# B&R Automation Studio project 8238 (part 19)

### history.Pkg_mnParam.txt
```
0.2.0	18.8.2011	- Import-Verzeichnis wird im Hochlauf gelöscht
			- Es werden auch REAL-Parameter unterstützt. (not tested)
0.3.0	24.8.2011	- IP-CSV-Rowtype ergänzt. (90)
0.4.0	01.09.2011	- Info_typ geändert. Es wird jetzt auch ausgegeben, welcher Container geändert wurde
0.5.0	20.09.2011	- mnParamStat und mnParamStatAd ergänzt.
			  Kapselung von Stati. z.B. xParamOK, dtExportContent
0.6.0	07.10.2011	- Maschinennummer wird aus _mnr.csv gelesen und in die _Info_-Struktur geschrieben
0.6.1	18.11.2011	- Liefert jetzt eine Fehlermeldung, wenn die zu importierende Datei keine Maschinennummer enthält
0.6.2	28.11.2011	- mnParamLib : mnParam_WritePVNum. UDINT wurde als UINT behandelt.
0.7.0	20.10.2011	- Umstellung auf AS 3.0.90
					- Berücksichtigung von WSTRING
					- utfMachineNumber und xParamOK in das IFmnParam.Out
0.8.0	20.12.2011	- Logging in das Logbuch der AR verlegt.
					- EXIT hinzugefügt.
					- Fehler im Init-Up behoben.
0.8.1	22.12.2011	- Severity für Log angepasst
0.8.2	02.01.2012	- Initialisierung der Text-Zeilen in GetCsvDat
					- Sprachdefinition ist 248, nicht 247
0.9.0	03.01.2012	- Packetversion in mnParamStatAd
0.9.1	10.01.2012	- Kommentar der Package-Version im Export wird dynamisch gelesen
0.10.0	18.01.2012	- Textzeilen werden jetzt mit bis zu 63 Zeichen ausgelesen
0.11.0	13.02.2012	- Speicherloch in der Initialisierung beseitigt. Beim Importieren vorhandener Datencontainer wurde Speicher nicht mehr frei gegeben.
0.11.1	15.02.2012	- Weiterentwicklung: Speicheroptimierung. Automatische Berechnung der Größe der Speicherpartition.
		16.02.2012	- Einführung von Funktionsbausteinen für Standardfunktionen.
					- Schreiben eines Inhaltsverzeichnisses von CSV-Datencontainerdateien im Exportverzeichnis
		17.02.2012	- Unit ist UINT
0.11.2	22.02.2012	- Helptext wurde auf 63 Zeichen begrenzt
					- Kompatibel zu hlKanLink 0.94.0
0.12.0	06.03.2012	- Kompatibel zu mnTest
0.12.1	08.03.2012	- Bugfix Editliste füllen
0.13.0	15.03.2012	- Editliste wird mit umgerechneten Werten gefüllt.
0.13.1	15.03.2012	- Ergänzt um die Anzahl der Nachkommastellen
					- Datenmodell erweitert um RefVisible und RefText
0.13.2	20.03.2012	- Abhängigkeiten ergänzt
0.13.9	20.03.2012	- Zwischenstand - Weiterentwicklung mnParam
0.14.0	21.03.2012	- Save-Editor und Delete indirect container implementiert. Bugfix im Delete Algorithmus auch für mnParamCmd
0.15.0	22.03.2012	- Zwischenversion. Es wird jetzt für das Edit-Feld nach Parameterindex, und nicht nach Container-Index gesucht.
					- Letzter Parameter eines Containers wurde nicht ausgelesen
					- Massenimport implementiert
					- Restore ist möglich
0.15.1	23.03.2012	- Maschinennummer des Datencontainers wird jetzt auch im Init-Up überprüft.
					- Die Überprüfung der Maschinennummer im zyklischen Teil kann applikativ deaktiviert werden.
					- Logger implementiert
					- Backup und Restore implementiert
0.16.0	23.03.2012	- Release
0.16.1	27.03.2012	- Bugfix: Container wurden im Init-Up nicht eingelesen
0.16.2	27.03.2012	- Weiterentwicklung
0.17.0	28.03.2012	- Namensliste für Instanzen kann gefüllt werden
					- Instanz NEU und KOPIEREN ist implementiert
0.17.1	29.03.2012	- Bugfix. Save Editor. Letzter Eintrag wurde nicht gesichert
0.18.0	29.03.2012	- Kategorie-Programm-Zuordnung ergänzt
0.18.1	30.03.2012	- Kategorie-Programm-Zuordnung um Kategorienamen erweitert
0.18.2	02.04.2012	- Kategoriedaten erweitert
0.19.0	03.04.2012	- Warnungen bei Importfehler
		04.04.2012	- _Info_ wird nicht mehr unterstützt
					- Bugfix: TOC wurde beim Import vom PC nicht aktualisiert
0.20.0	05.04.2012	- Die Quelle zum Füllen der Namensliste wird nur initial von den Konstanten übernommen.
					  Per Befehl kann die Quelle geändert werden.
0.20.1	10.04.2012	- Wenn die Dateien im Exportverzeichnis gelöscht wurden, hat der Parametermanager diese nicht
					  neu angelegt.
0.20.2	11.04.2012	- Maschinennummer mit Länge 0 wird als Fehler abgefangen
0.20.3	11.04.2012	- Ungültige Maschinennummer "dummy" als Konstante MNPARAM_INVALID_MACHINENO eingeführt
0.20.4	13.04.2012	- Warnung wird angezeigt, wenn der Parametermanager nicht bereit ist.
0.20.5	16.04.2012	- Beim Füllen des Editors, wurden die Parameter für die Namensliste zurückgesetzt
0.20.6	17.04.2012	- Es konnten keine Instanzen aus dem Editor gesichert werden. Der Pointer auf die StrucRoot wurde nicht ermittelt.
0.20.7	18.04.2012  - Instanz-Datenobjekte werden im Init teilweise wieder gelöscht.
					- In der Instanznamensliste werden noch die Instanznummern vorangestellt
0.21.0	23.04.2012	- Wir create instance oder copy instance eine negative Instanznummer übergeben, wird die nächste freie Instanz angelegt
					- Bei Fill Namelist wird automatisch die Category-Program-Cache-Liste aktualisiert
0.21.1	23.04.2012	- Copy hat nicht funktioniert
0.22.0	11.05.2012	- Restore lädt auch den cpcache
0.23.0	04.06.2012	- Im InitUp werden beim Importieren der Container auf jeden Falle vorher alle Daten auf Default gesetzt.
					- Wird nach dem Hochlauf ein USB-Stick mit dem Unterverzeichnis SetupKG erkannt, dann wird das Userverzeichnis entsprechend
					  überschrieben
					- Die Struktur "Machinestate" wird nicht mehr unterstützt
0.24.0 12.06.2012	- Beim Import von Parametern werden numerische Parameter auf ihre min- und max-Werte begrenzt.
					- Hilfstexte für Parameter auf 255 Zeichen erweitert.
					- Im Parametereditor kann nun gesteuert werden, ob Funktions- und Instanztexte in den Parametertext eingefügt werden.
					  Zusätzlich wird der Funktionstext und Instanztext zum Parameter separat ausgegeben. Parameter können nach Funktionen
					  gefiltert werden
0.24.1	26.06.2012	- Warnung unterdrückt
0.24.2	17.07.2012	- Filehandles wurden nach FileCreate nicht freigegeben.
0.24.3	03.09.2012	- Bugfix: Bug 835 - Kopierte Datencontainer sind schreibgeschützt. Behoben
0.25.0	06.09.2012	- Erweiterung Bug 821: Neue Konstante: MNPARAM_REQMISSINGMNO vom Typ USINT
					  0 : Wenn die Datei _mnr.csv fehlt, wird die Maschinennummer "dummy" gesetzt.
					  1 : Wenn die Datei _mnr.csv fehlt, erwartet der Parametermanager über das Interface IFmnParam
					  	  das Setzen der Maschinennummer in IFmnParam.In.utfSetMachineNumber. Danach muss die Strukturvariable
						  IFmnParam.In.xSetMachnineNumber auf TRUE gesetzt werden. Die _mnr.csv wird erzeugt und die Steuerung wird
						  neu gestartet.
```

### CfgMsgStat.mnParam.txt
```
;****************************
; Parameter Manager
;*****************************
00001, 00001, 00000, 00000;
00001, 00002, 00000, 00000;
00001, 00003, 00000, 00000;
00001, 00004, 00000, 00000;
00001, 00005, 00000, 00000;
00001, 00006, 00000, 00000;
00001, 00007, 00000, 00000;
00001, 00009, 00000, 00000;
00001, 20000, 00000, 00000;
```

### Package Logical/Standard/Kanlink/KGFramework/Pkg_mnTxt - Text-Manager

### Pkg_mnTxt.typ - Global data types
```iecst
(********************************************************************
 * COPYRIGHT -- Herbert Kannegiesser GmbH
 ********************************************************************
 * Package: Pkg_mnTxt
 * File: Pkg_mnTxt.typ
 * Author: hunholz
 * Created: November 25, 2011
 ********************************************************************
 * Data types of package Pkg_mnTxt
 ********************************************************************)
(*Interface*)

TYPE
	IFmnTxt_Typ : 	STRUCT
		In : IFmnTxt_In_Typ;
		Out : IFmnTxt_Out_Typ;
	END_STRUCT;
	IFmnTxt_Out_Typ : 	STRUCT
		wSelectedLanguage : UINT; (*Aktive Sprache*)
		wSelectLanguageStatus : UINT; (*0 - Sprache gültig, nur dann sind auch die Pointer auf die Texte gültig
60000..65000 - Fehler
65535 - Sprache wird geladen*)
		wLCIDs : ARRAY[0..MNTXT_MAX_IDX_LCID]OF UINT;
		wCntLCID : UINT;
		wCntInstanceTxt : UINT := 0;
		wCntFunctionTxt : UINT := 0;
		wCntParamTxt : UINT := 0;
		wCntParamHlpTxt : UINT := 0;
		wCntMessageTxt : UINT := 0;
		wCntMessageHlpTxt : UINT := 0;
		ptrInstanceTxtList : UDINT; (*Zeigt auf das Datenobjekt _mnTxtI, Zeilen vom Typ mnTxt_TxtLine_Typ*)
		ptrFunctionTxtList : UDINT; (*Zeigt auf das Datenobjekt _mnTxtF, Zeilen vom Typ mnTxt_TxtLine_Typ*)
		ptrParamTxtList : UDINT; (*Zeigt auf das Datenobjekt _mnTxtP, Zeilen vom Typ mnTxt_TxtLine_Typ*)
		ptrParamHelpTxtList : UDINT; (*Zeigt auf das Datenobjekt _mnTxtPh, Zeilen vom Typ mnTxt_HelpTxtLine_Typ*)
		ptrMessageTxtList : UDINT; (*Zeigt auf das Datenobjekt _mnTxtM, Zeilen vom Typ mnTxt_TxtLine_Typ*)
		ptrMessageHelpTxtList : UDINT; (*Zeigt auf das Datenobjekt _mnTxtMh, Zeilen vom Typ mnTxt_HelpTxtLine_Typ*)
	END_STRUCT;
	IFmnTxt_In_Typ : 	STRUCT
		wSelectLanguage : UINT; (*LCID der Sprache, die genutzt werden soll*)
	END_STRUCT;
END_TYPE

(*Parameter*)

TYPE
	mnTxtPar_Typ : 	STRUCT
		Mac : mnTxtPar_Mac_Typ; (*Maschinenparameter*)
	END_STRUCT;
	mnTxtPar_Mac_Typ : 	STRUCT
		wStartUpLanguage : UINT := 0; (*Die Sprache ist remanent. Ist hier ein Wert > 0 gewählt, wird diese Sprache beim Einschalten immer geladen.*)
	END_STRUCT;
END_TYPE

(*Status*)

TYPE
	mnTxtStatAd_Typ : 	STRUCT
		sPkgVersion : STRING[10];
	END_STRUCT;
END_TYPE

(*Öffentliche Typen*)

TYPE
	mnTxt_TxtLine_Typ : 	STRUCT
		wFunctionID : UINT; (*Funktions-Identifier*)
		wNumber : UINT; (*Textnummer*)
		wInstance : UINT; (*Instanznummer, um kompatibel zu mnMsg zu sein*)
		utfText : WSTRING[63]; (*Eigentlicher Text*)
	END_STRUCT;
	mnTxt_HelpTxtLine_Typ : 	STRUCT
		wFunctionID : UINT; (*Funktions-Identifier*)
		wNumber : UINT; (*Textnummer*)
		wInstance : UINT; (*Instanznummer, um kompatibel zu mnMsg zu sein*)
		utfText : WSTRING[255]; (*Eigentlicher Hilfstext*)
	END_STRUCT;
END_TYPE
```

### Pkg_mnTxt.var - Global variables
```iecst
(********************************************************************
 * COPYRIGHT -- Herbert Kannegiesser GmbH
 ********************************************************************
 * Package: Pkg_mnTxt
 * File: Pkg_mnTxt.var
 * Author: hunholz
 * Created: November 25, 2011
 ********************************************************************
 * Variables of package Pkg_mnTxt
 ********************************************************************)
(*KONSTANTEN*)
VAR CONSTANT
	MNTXT_DATOBJNAME_INSTXT : STRING[11] := '_mnTxtI'; (*Name des Datenmoduls, in dem die Instanztexte abgelegt sind*)
	MNTXT_DATOBJNAME_FUNTXT : STRING[11] := '_mnTxtF'; (*Name des Datenmoduls, in dem die Funktionstexte abgelegt sind*)
	MNTXT_DATOBJNAME_PARTXT : STRING[11] := '_mnTxtP'; (*Name des Datenmoduls, in dem die Parametertexte abgelegt sind*)
	MNTXT_DATOBJNAME_PARHELPTXT : STRING[11] := '_mnTxtPh'; (*Name des Datenmoduls, in dem die Parameterhilfstexte abgelegt sind*)
	MNTXT_DATOBJNAME_MSGTXT : STRING[11] := '_mnTxtM'; (*Name des Datenmoduls, in dem die Meldungstexte abgelegt sind*)
	MNTXT_DATOBJNAME_MSGHELPTXT : STRING[11] := '_mnTxtMh'; (*Name des Datenmoduls, in dem die Meldungshilfstexte abgelegt sind*)
END_VAR
(*-- LCID --*)
VAR CONSTANT
	MNTXT_LCID_GERMAN : UINT := 1031; (*LCID German*)
	MNTXT_LCID_ENGLISH_US : UINT := 1033; (*LCID English USA*)
END_VAR
(*-- Stati --*)
VAR CONSTANT
	MNTXT_STAT_OK : UINT := 0;
	MNTXT_STAT_NOLANGUAGE : UINT := 1; (*Keine gültige Sprache geladen*)
	MNTXT_STAT_INIT : UINT := 100;
	MNTXT_STAT_ERRDATOBJ : UINT := 60000; (*Datenobjekte für Texte konnten nicht erstellt werden.*)
	MNTXT_STAT_ERRMSGCFG : UINT := 60001; (*Message-Config Fehler*)
	MNTXT_STAT_ERRMEM : UINT := 60002; (*Speicher nicht allokierbar oder nicht ausreichend*)
	MNTXT_STAT_ERRLCID : UINT := 60003; (*Fehler beim laden von LCID.csv*)
	MNTXT_STAT_ERRFUNCTIONTXT : UINT := 60004;
	MNTXT_STAT_ERRINSTANCETXT : UINT := 60005;
	MNTXT_STAT_ERRMESSAGETXT : UINT := 60006;
	MNTXT_STAT_ERRPARAMTXT : UINT := 60007;
	MNTXT_STAT_LOADING : UINT := 65535;
END_VAR
(*Interface*)
VAR
	IFmnTxt : IFmnTxt_Typ;
END_VAR
(*Status*)
VAR
	mnTxtStatAd : mnTxtStatAd_Typ;
END_VAR
(*Parameter*)
VAR
	mnTxtPar : mnTxtPar_Typ;
END_VAR
```

### Program Logical/Standard/Kanlink/KGFramework/Pkg_mnTxt/mnTxt (IEC) - Text-Manager

#### mnTxtCyclic.st - Cyclic code
```iecst
(********************************************************************
 * COPYRIGHT -- Herbert Kannegiesser GmbH
 ********************************************************************
 * Program: mnTxt
 * File: mnTxtCyclic.st
 * Author: hunholz
 * Created: November 25, 2011
 ********************************************************************
 * Implementation of program mnTxt
 ********************************************************************)

PROGRAM _CYCLIC

	// Auf Sprachwechsel reagieren, bzw. letzte Sprache laden

	IF _xInitOK THEN

		IF IFmnTxt.Out.wSelectLanguageStatus = MNTXT_STAT_OK THEN

			// Sprache kann neu gewählt werden
			IF _wActLCID <> IFmnTxt.In.wSelectLanguage AND IFmnTxt.In.wSelectLanguage <> 0 THEN

				_wIdxLCID := 0;

				REPEAT

					IF IFmnTxt.In.wSelectLanguage = IFmnTxt.Out.wLCIDs[_wIdxLCID] THEN

						_wActLCID := IFmnTxt.In.wSelectLanguage;

						IFmnTxt.Out.wSelectedLanguage := _wActLCID;
						IFmnTxt.Out.wSelectLanguageStatus := MNTXT_STAT_LOADING;
						_LoadState := _ls_load_functiontxt_01;

					END_IF

					_wIdxLCID := _wIdxLCID + 1;

					UNTIL
					_wActLCID = IFmnTxt.In.wSelectLanguage OR _wIdxLCID >= IFmnTxt.Out.wCntLCID OR _wIdxLCID > MNTXT_MAX_IDX_LCID
				END_REPEAT

			END_IF

		ELSIF IFmnTxt.Out.wSelectLanguageStatus = MNTXT_STAT_NOLANGUAGE THEN

			IF _LoadState = _ls_idle THEN

				// Sprache erstmals laden
				IF _wActLCID = 0 THEN

					IF _xGermanExist THEN

						_wActLCID := MNTXT_LCID_GERMAN;

					ELSE

						_wActLCID := IFmnTxt.Out.wLCIDs[0];

					END_IF

				END_IF

				IFmnTxt.Out.wSelectedLanguage := _wActLCID;
				IFmnTxt.Out.wSelectLanguageStatus := MNTXT_STAT_LOADING;
				_LoadState := _ls_load_functiontxt_01;

			END_IF

		END_IF

	END_IF

	// Zyklusbegrenzung zurücksetzen

	_lCycleCounter := 0;

	// Statemachine

	CASE _LoadState OF

		_ls_idle:

		// Grundzustand, nichts tun

		//###########################################################################################
		// FUNKTIONSTEXTE LADEN
		//###########################################################################################

		_ls_load_functiontxt_01:

			// Nachsehen, ob Funktionstexte existieren

			IFmnTxt.Out.wCntFunctionTxt := 0;

			IF MNTXT_LOAD_FUNCTIONTEXT AND _CheckDoFunc.doId <> 0 THEN

				IF MNTXT_ENABLE_LANSPECRESOURCE = 1 THEN

					_sLCID := UINT_TO_STRING(_wActLCID);
					_sPath := CONCAT('Language\Function',_sLCID);
					_sPath := CONCAT(_sPath,'.csv');

				ELSE

					_sPath := 'Language\Function.csv';

				END_IF

				_FileInfo(enable := TRUE, pDevice := ADR(KG_DEVICE_COMPACTFLASH), pName := ADR(_sPath), pInfo := ADR(_fiFileInfo));

				IF _FileInfo.status = ERR_OK THEN

					_LoadState := _ls_load_functiontxt_02;

				ELSIF _FileInfo.status <> ERR_FUB_BUSY THEN

					_LoadState := _ls_load_instancetxt_01;

				END_IF

			ELSE

				_LoadState := _ls_load_instancetxt_01;

			END_IF

		_ls_load_functiontxt_02:

			// Speicher zum Parsen der Funktionstexte allokieren
			_MemPartAlloc(enable := TRUE, ident := _MemPartCreate.ident, len := _fiFileInfo.size-SIZEOF(KGBOM) );

			IF _MemPartAlloc.status = ERR_OK THEN

				_lAdrFile := _MemPartAlloc.mem;
				_LoadState := _ls_load_functiontxt_03;

			ELSIF _MemPartAlloc.status <> ERR_FUB_BUSY THEN

				IFmnTxt.Out.wSelectLanguageStatus := MNTXT_STAT_ERRMEM;
				_LoadState := _ls_error;

			END_IF

		_ls_load_functiontxt_03:

			_FileOpen(enable := TRUE, pDevice := ADR(KG_DEVICE_COMPACTFLASH), pFile := ADR(_sPath), mode := fiREAD_ONLY);

			IF _FileOpen.status = ERR_OK THEN

				_LoadState := _ls_load_functiontxt_04;

			ELSIF _FileOpen.status <> ERR_FUB_BUSY THEN

				IFmnTxt.Out.wSelectLanguageStatus := MNTXT_STAT_ERRFUNCTIONTXT;
				_LoadState := _ls_error;

			END_IF

		_ls_load_functiontxt_04:

			_FileRead(enable := TRUE, ident := _FileOpen.ident, offset := SIZEOF(KGBOM),pDest := _lAdrFile, len :=  _fiFileInfo.size-SIZEOF(KGBOM) );

			IF _FileRead.status <> ERR_FUB_BUSY THEN

				_LoadState := _ls_load_functiontxt_05;

			END_IF

		_ls_load_functiontxt_05:

			_FileClose(enable := TRUE, ident := _FileOpen.ident);

			IF _FileClose.status <> ERR_FUB_BUSY THEN

				IF _FileRead.status = ERR_OK THEN

					_LoadState := _ls_load_functiontxt_06;

				ELSE
					IFmnTxt.Out.wSelectLanguageStatus := MNTXT_STAT_ERRFUNCTIONTXT;
					_LoadState := _ls_error;

				END_IF

			END_IF

		_ls_load_functiontxt_06:

			// Zeilen in der Datei zählen und Startadressen ermitteln

			_CountLines.enable := TRUE;
			_CountLines.pFile := _lAdrFile;
			_CountLines.FileSize := _fiFileInfo.size - SIZEOF(KGBOM);
			_CountLines.MaxLines := MNTXT_MAXPARSELINES;
			_CountLines.pAdresses := _lAdrLineAdress;
			_CountLines.pLens := _lAdrLineLen;

			_CountLines();

			IF _CountLines.status = ERR_OK THEN

				_LoadState := _ls_load_functiontxt_07;

				_wStartLine := 1;
				_wIdxFunctionTxt := 0;
				_GetCsvDat.enable := TRUE;

			ELSE

				IFmnTxt.Out.wSelectLanguageStatus := MNTXT_STAT_ERRFUNCTIONTXT;
				_LoadState := _ls_error;

			END_IF

		_ls_load_functiontxt_07:

			// Datei parsen

			REPEAT

				brwcsncpy( ADR(_GetCsvDat.utfCsvString), _plLineAdress[_wStartLine], MIN(299, _pwLineLen[_wStartLine]));
				_GetCsvDat();
				_wStartLine := _wStartLine + 1;

				IF _GetCsvDat.RowType = 200 AND _GetCsvDat.csvTextRow.LCID = _wActLCID THEN

					_TxtLine.wNumber := 0;
					_TxtLine.wFunctionID := _GetCsvDat.csvTextRow.FunctionID;
					_TxtLine.utfText := _GetCsvDat.csvTextRow.utfText;

					_dowFuncTxt(enable := TRUE, ident := _CheckDoFunc.doId, Offset := SIZEOF(_TxtLine)*_wIdxFunctionTxt, pSource := ADR(_TxtLine), len := SIZEOF(_TxtLine));

					_wIdxFunctionTxt := _wIdxFunctionTxt + 1;

				END_IF

				_lCycleCounter := _lCycleCounter + 1;

				UNTIL

				_lCycleCounter > 20 OR _wIdxFunctionTxt > MNTXT_MAX_IDX_TXT_FUNCTION OR _wStartLine > _CountLines.CntLines

			END_REPEAT

			IF _wIdxFunctionTxt > MNTXT_MAX_IDX_TXT_FUNCTION OR _wStartLine > _CountLines.CntLines THEN

				IFmnTxt.Out.wCntFunctionTxt := _wIdxFunctionTxt;
				_LoadState := _ls_load_functiontxt_08;

			END_IF

		_ls_load_functiontxt_08:

			// Speicher frei geben

			_MemPartFree(enable := TRUE, ident := _MemPartCreate.ident, mem := _lAdrFile);

			IF _MemPartFree.status = ERR_OK THEN

				_LoadState := _ls_load_instancetxt_01;

			ELSIF _MemPartFree.status <> ERR_FUB_BUSY THEN

				IFmnTxt.Out.wSelectLanguageStatus := MNTXT_STAT_ERRFUNCTIONTXT;
				_LoadState := _ls_error;

			END_IF

		//###########################################################################################
		// INSTANZTEXTE LADEN
		//###########################################################################################

		_ls_load_instancetxt_01:

			// Nachsehen, ob Instanztexte existieren

			IFmnTxt.Out.wCntInstanceTxt := 0;

			IF MNTXT_LOAD_INSTANCETEXT AND _CheckDoInst.doId <> 0 THEN

				IF MNTXT_ENABLE_LANSPECRESOURCE = 1 THEN

					_sLCID := UINT_TO_STRING(_wActLCID);
					_sPath := CONCAT('Language\Instance',_sLCID);
					_sPath := CONCAT(_sPath,'.csv');

				ELSE

					_sPath := 'Language\Instance.csv';

				END_IF

				_FileInfo(enable := TRUE, pDevice := ADR(KG_DEVICE_COMPACTFLASH), pName := ADR(_sPath), pInfo := ADR(_fiFileInfo));

				IF _FileInfo.status = ERR_OK THEN

					_LoadState := _ls_load_instancetxt_02;

				ELSIF _FileInfo.status <> ERR_FUB_BUSY THEN

					_LoadState := _ls_load_messagetxt_01;

				END_IF

			ELSE

				_LoadState := _ls_load_messagetxt_01;

			END_IF

		_ls_load_instancetxt_02:

			// Speicher zum Parsen der Funktionstexte allokieren
			_MemPartAlloc(enable := TRUE, ident := _MemPartCreate.ident, len := _fiFileInfo.size-SIZEOF(KGBOM) );

			IF _MemPartAlloc.status = ERR_OK THEN

				_lAdrFile := _MemPartAlloc.mem;
				_LoadState := _ls_load_instancetxt_03;

			ELSIF _MemPartAlloc.status <> ERR_FUB_BUSY THEN

				IFmnTxt.Out.wSelectLanguageStatus := MNTXT_STAT_ERRMEM;
				_LoadState := _ls_error;

			END_IF

		_ls_load_instancetxt_03:

			_FileOpen(enable := TRUE, pDevice := ADR(KG_DEVICE_COMPACTFLASH), pFile := ADR(_sPath), mode := fiREAD_ONLY);

			IF _FileOpen.status = ERR_OK THEN

				_LoadState := _ls_load_instancetxt_04;

			ELSIF _FileOpen.status <> ERR_FUB_BUSY THEN

				IFmnTxt.Out.wSelectLanguageStatus := MNTXT_STAT_ERRINSTANCETXT;
				_LoadState := _ls_error;

			END_IF

		_ls_load_instancetxt_04:

			_FileRead(enable := TRUE, ident := _FileOpen.ident, offset := SIZEOF(KGBOM),pDest := _lAdrFile, len :=  _fiFileInfo.size-SIZEOF(KGBOM) );

			IF _FileRead.status <> ERR_FUB_BUSY THEN

				_LoadState := _ls_load_instancetxt_05;

			END_IF

		_ls_load_instancetxt_05:

			_FileClose(enable := TRUE, ident := _FileOpen.ident);

			IF _FileClose.status <> ERR_FUB_BUSY THEN

				IF _FileRead.status = ERR_OK THEN

					_LoadState := _ls_load_instancetxt_06;

				ELSE
					IFmnTxt.Out.wSelectLanguageStatus := MNTXT_STAT_ERRINSTANCETXT;
					_LoadState := _ls_error;

				END_IF

			END_IF

		_ls_load_instancetxt_06:

			// Zeilen in der Datei zählen und Startadressen ermitteln

			_CountLines.enable := TRUE;
			_CountLines.pFile := _lAdrFile;
			_CountLines.FileSize := _fiFileInfo.size - SIZEOF(KGBOM);
			_CountLines.MaxLines := MNTXT_MAXPARSELINES;
			_CountLines.pAdresses := _lAdrLineAdress;
			_CountLines.pLens := _lAdrLineLen;

			_CountLines();

			IF _CountLines.status = ERR_OK THEN

				_LoadState := _ls_load_instancetxt_07;

				_wStartLine := 1;
				_wIdxInstanceTxt := 0;
				_GetCsvDat.enable := TRUE;

			ELSE

				IFmnTxt.Out.wSelectLanguageStatus := MNTXT_STAT_ERRINSTANCETXT;
				_LoadState := _ls_error;

			END_IF

		_ls_load_instancetxt_07:

			// Datei parsen

			REPEAT

				brwcsncpy( ADR(_GetCsvDat.utfCsvString), _plLineAdress[_wStartLine], MIN(299, _pwLineLen[_wStartLine]));
				_GetCsvDat();
				_wStartLine := _wStartLine + 1;

				IF _GetCsvDat.RowType = 200 AND _GetCsvDat.csvTextRow.LCID = _wActLCID THEN

					_TxtLine.wNumber := _GetCsvDat.csvTextRow.TextNo;
					_TxtLine.wFunctionID := _GetCsvDat.csvTextRow.FunctionID;
					_TxtLine.utfText := _GetCsvDat.csvTextRow.utfText;

					_dowInstTxt(enable := TRUE, ident := _CheckDoInst.doId, Offset := SIZEOF(_TxtLine)*_wIdxInstanceTxt, pSource := ADR(_TxtLine), len := SIZEOF(_TxtLine));

					_wIdxInstanceTxt := _wIdxInstanceTxt + 1;

				END_IF

				_lCycleCounter := _lCycleCounter + 1;

				UNTIL

				_lCycleCounter > 20 OR _wIdxInstanceTxt > MNTXT_MAX_IDX_TXT_INSTANCE OR _wStartLine > _CountLines.CntLines

			END_REPEAT

			IF _wIdxInstanceTxt > MNTXT_MAX_IDX_TXT_INSTANCE OR _wStartLine > _CountLines.CntLines THEN

				IFmnTxt.Out.wCntInstanceTxt := _wIdxInstanceTxt;
				_LoadState := _ls_load_instancetxt_08;

			END_IF

		_ls_load_instancetxt_08:

			// Speicher frei geben

			_MemPartFree(enable := TRUE, ident := _MemPartCreate.ident, mem := _lAdrFile);

			IF _MemPartFree.status = ERR_OK THEN

				_LoadState := _ls_load_messagetxt_01;

			ELSIF _MemPartFree.status <> ERR_FUB_BUSY THEN

				IFmnTxt.Out.wSelectLanguageStatus := MNTXT_STAT_ERRINSTANCETXT;
				_LoadState := _ls_error;

			END_IF

		//###########################################################################################
		// MELDUNGSTEXTE LADEN
		//###########################################################################################

		_ls_load_messagetxt_01:

			// Nachsehen, ob Meldungstexte existieren

			IFmnTxt.Out.wCntMessageTxt := 0;
			IFmnTxt.Out.wCntMessageHlpTxt := 0;

			IF MNTXT_ENABLE_LANSPECRESOURCE = 1 THEN

				_sLCID := UINT_TO_STRING(_wActLCID);
				_sPath := CONCAT('Messages\Messages',_sLCID);
				_sPath := CONCAT(_sPath,'.csv');

			ELSE

				_sPath := 'Messages\Messages.csv';

			END_IF

			_FileInfo(enable := TRUE, pDevice := ADR(KG_DEVICE_COMPACTFLASH), pName := ADR(_sPath), pInfo := ADR(_fiFileInfo));

			IF _FileInfo.status = ERR_OK THEN

				_LoadState := _ls_load_messagetxt_02;

			ELSIF _FileInfo.status <> ERR_FUB_BUSY THEN

				IFmnTxt.Out.wSelectLanguageStatus := MNTXT_STAT_ERRMESSAGETXT;
				_LoadState := _ls_error;

			END_IF

		_ls_load_messagetxt_02:

			// Speicher zum Parsen der Funktionstexte allokieren
			_MemPartAlloc(enable := TRUE, ident := _MemPartCreate.ident, len := _fiFileInfo.size-SIZEOF(KGBOM) );

			IF _MemPartAlloc.status = ERR_OK THEN

				_lAdrFile := _MemPartAlloc.mem;
				_LoadState := _ls_load_messagetxt_03;

			ELSIF _MemPartAlloc.status <> ERR_FUB_BUSY THEN

				IFmnTxt.Out.wSelectLanguageStatus := MNTXT_STAT_ERRMEM;
				_LoadState := _ls_error;

			END_IF

		_ls_load_messagetxt_03:

			_FileOpen(enable := TRUE, pDevice := ADR(KG_DEVICE_COMPACTFLASH), pFile := ADR(_sPath), mode := fiREAD_ONLY);

			IF _FileOpen.status = ERR_OK THEN

				_LoadState := _ls_load_messagetxt_04;

			ELSIF _FileOpen.status <> ERR_FUB_BUSY THEN

				IFmnTxt.Out.wSelectLanguageStatus := MNTXT_STAT_ERRMESSAGETXT;
				_LoadState := _ls_error;

			END_IF

		_ls_load_messagetxt_04:

			_FileRead(enable := TRUE, ident := _FileOpen.ident, offset := SIZEOF(KGBOM),pDest := _lAdrFile, len :=  _fiFileInfo.size-SIZEOF(KGBOM) );

			IF _FileRead.status <> ERR_FUB_BUSY THEN

				_LoadState := _ls_load_messagetxt_05;

			END_IF

		_ls_load_messagetxt_05:

			_FileClose(enable := TRUE, ident := _FileOpen.ident);

			IF _FileClose.status <> ERR_FUB_BUSY THEN

				IF _FileRead.status = ERR_OK THEN

					_LoadState := _ls_load_messagetxt_06;

				ELSE
					IFmnTxt.Out.wSelectLanguageStatus := MNTXT_STAT_ERRMESSAGETXT;
					_LoadState := _ls_error;

				END_IF

			END_IF

		_ls_load_messagetxt_06:

			// Zeilen in der Datei zählen und Startadressen ermitteln

			_CountLines.enable := TRUE;
			_CountLines.pFile := _lAdrFile;
			_CountLines.FileSize := _fiFileInfo.size - SIZEOF(KGBOM);
			_CountLines.MaxLines := MNTXT_MAXPARSELINES;
			_CountLines.pAdresses := _lAdrLineAdress;
			_CountLines.pLens := _lAdrLineLen;

			_CountLines();

			IF _CountLines.status = ERR_OK THEN

				_LoadState := _ls_load_messagetxt_07;

				_wStartLine := 1;
				_wIdxMessageTxt := 0;
				_wIdxMessageHelpTxt := 0;
				_GetCsvDat.enable := TRUE;

			ELSE

				IFmnTxt.Out.wSelectLanguageStatus := MNTXT_STAT_ERRMESSAGETXT;
				_LoadState := _ls_error;

			END_IF

		_ls_load_messagetxt_07:

			// Datei parsen

			REPEAT

				brwcsncpy( ADR(_GetCsvDat.utfCsvString), _plLineAdress[_wStartLine], MIN(299, _pwLineLen[_wStartLine]));
				_GetCsvDat();
				_wStartLine := _wStartLine + 1;

				IF _GetCsvDat.RowType = 200 AND _GetCsvDat.csvTextRow.LCID = _wActLCID AND _wIdxMessageTxt < _lLenMsg THEN

					_TxtLine.wNumber := _GetCsvDat.csvTextRow.TextNo;
					_TxtLine.wFunctionID := _GetCsvDat.csvTextRow.FunctionID;
					_TxtLine.utfText := _GetCsvDat.csvTextRow.utfText;

					_dowMsgTxt(enable := TRUE, ident := _CheckDoMsg.doId, Offset := SIZEOF(_TxtLine)*_wIdxMessageTxt, pSource := ADR(_TxtLine), len := SIZEOF(_TxtLine));

					_wIdxMessageTxt := _wIdxMessageTxt + 1;

				ELSIF _GetCsvDat.RowType = 210 AND _GetCsvDat.csvHelpTextRow.LCID = _wActLCID AND _wIdxMessageHelpTxt < _lLenMsg THEN

					_TxtHelpLine.wNumber := _GetCsvDat.csvHelpTextRow.TextNo;
					_TxtHelpLine.wFunctionID := _GetCsvDat.csvHelpTextRow.FunctionID;

					_utfRC(pInput := ADR(_GetCsvDat.csvHelpTextRow.utfHelpText), pOutput := ADR(_TxtHelpLine.utfText), lSizeOutput := SIZEOF(_TxtHelpLine.utfText), xWSTRING := TRUE);

//					_TxtHelpLine.utfText := _GetCsvDat.csvHelpTextRow.utfHelpText;

					_dowMsgHlpTxt(enable := TRUE, ident := _CheckDoMsgHlp.doId, Offset := SIZEOF(_TxtHelpLine)*_wIdxMessageHelpTxt, pSource := ADR(_TxtHelpLine), len := SIZEOF(_TxtHelpLine));

					_wIdxMessageHelpTxt := _wIdxMessageHelpTxt + 1;

				END_IF

				_lCycleCounter := _lCycleCounter + 1;

				UNTIL

				_lCycleCounter > 20 OR (_wIdxMessageTxt >= _lLenMsg AND _wIdxMessageHelpTxt >= _lLenMsg) OR _wStartLine > _CountLines.CntLines

			END_REPEAT

			IF (_wIdxMessageTxt >= _lLenMsg AND _wIdxMessageHelpTxt >= _lLenMsg) OR _wStartLine > _CountLines.CntLines THEN

				IFmnTxt.Out.wCntMessageTxt := _wIdxMessageTxt;
				IFmnTxt.Out.wCntMessageHlpTxt := _wIdxMessageHelpTxt;
				_LoadState := _ls_load_messagetxt_08;

			END_IF

		_ls_load_messagetxt_08:

			// Speicher frei geben

			_MemPartFree(enable := TRUE, ident := _MemPartCreate.ident, mem := _lAdrFile);

			IF _MemPartFree.status = ERR_OK THEN

				_LoadState := _ls_load_paramtxt_01;

			ELSIF _MemPartFree.status <> ERR_FUB_BUSY THEN

				IFmnTxt.Out.wSelectLanguageStatus := MNTXT_STAT_ERRMESSAGETXT;
				_LoadState := _ls_error;

			END_IF

		//###########################################################################################
		// PARAMETERTEXTE LADEN
		//###########################################################################################

		_ls_load_paramtxt_01:

			// Nachsehen, ob Parametertexte existieren

			IFmnTxt.Out.wCntParamTxt := 0;
			IFmnTxt.Out.wCntParamHlpTxt := 0;

			IF MNTXT_LOAD_PARAMETERTEXT AND _CheckDoPar.doId <> 0 THEN

				IF MNTXT_ENABLE_LANSPECRESOURCE = 1 THEN

					_sLCID := UINT_TO_STRING(_wActLCID);
					_sPath := CONCAT('Language\ParamTxt',_sLCID);
					_sPath := CONCAT(_sPath,'.csv');

				ELSE

					_sPath := 'Language\ParamTxt.csv';

				END_IF

				_FileInfo(enable := TRUE, pDevice := ADR(KG_DEVICE_COMPACTFLASH), pName := ADR(_sPath), pInfo := ADR(_fiFileInfo));

				IF _FileInfo.status = ERR_OK THEN

					_LoadState := _ls_load_paramtxt_02;

				ELSIF _FileInfo.status <> ERR_FUB_BUSY THEN

					IFmnTxt.Out.wSelectLanguageStatus := MNTXT_STAT_ERRPARAMTXT;
					_LoadState := _ls_error;

				END_IF

			ELSE

				_LoadState := _ls_idle;
				IFmnTxt.Out.wSelectLanguageStatus := MNTXT_STAT_OK;

			END_IF

		_ls_load_paramtxt_02:

			// Speicher zum Parsen der Parametertexte allokieren
			_MemPartAlloc(enable := TRUE, ident := _MemPartCreate.ident, len := _fiFileInfo.size-SIZEOF(KGBOM) );

			IF _MemPartAlloc.status = ERR_OK THEN

				_lAdrFile := _MemPartAlloc.mem;
				_LoadState := _ls_load_paramtxt_03;

			ELSIF _MemPartAlloc.status <> ERR_FUB_BUSY THEN

				IFmnTxt.Out.wSelectLanguageStatus := MNTXT_STAT_ERRMEM;
				_LoadState := _ls_error;

			END_IF

		_ls_load_paramtxt_03:

			_FileOpen(enable := TRUE, pDevice := ADR(KG_DEVICE_COMPACTFLASH), pFile := ADR(_sPath), mode := fiREAD_ONLY);

			IF _FileOpen.status = ERR_OK THEN

				_LoadState := _ls_load_paramtxt_04;

			ELSIF _FileOpen.status <> ERR_FUB_BUSY THEN

				IFmnTxt.Out.wSelectLanguageStatus := MNTXT_STAT_ERRPARAMTXT;
				_LoadState := _ls_error;

			END_IF

		_ls_load_paramtxt_04:

			_FileRead(enable := TRUE, ident := _FileOpen.ident, offset := SIZEOF(KGBOM),pDest := _lAdrFile, len :=  _fiFileInfo.size-SIZEOF(KGBOM) );

			IF _FileRead.status <> ERR_FUB_BUSY THEN

				_LoadState := _ls_load_paramtxt_05;

			END_IF

		_ls_load_paramtxt_05:

			_FileClose(enable := TRUE, ident := _FileOpen.ident);

			IF _FileClose.status <> ERR_FUB_BUSY THEN

				IF _FileRead.status = ERR_OK THEN

					_LoadState := _ls_load_paramtxt_06;

				ELSE
					IFmnTxt.Out.wSelectLanguageStatus := MNTXT_STAT_ERRPARAMTXT;
					_LoadState := _ls_error;

				END_IF

			END_IF

		_ls_load_paramtxt_06:

			// Zeilen in der Datei zählen und Startadressen ermitteln

			_CountLines.enable := TRUE;
			_CountLines.pFile := _lAdrFile;
			_CountLines.FileSize := _fiFileInfo.size - SIZEOF(KGBOM);
			_CountLines.MaxLines := MNTXT_MAXPARSELINES;
			_CountLines.pAdresses := _lAdrLineAdress;
			_CountLines.pLens := _lAdrLineLen;

			_CountLines();

			IF _CountLines.status = ERR_OK THEN

				_LoadState := _ls_load_paramtxt_07;

				_wStartLine := 1;
				_wIdxParamTxt := 0;
				_wIdxParamHelpTxt := 0;
				_GetCsvDat.enable := TRUE;

			ELSE

				IFmnTxt.Out.wSelectLanguageStatus := MNTXT_STAT_ERRPARAMTXT;
				_LoadState := _ls_error;

			END_IF

		_ls_load_paramtxt_07:

			// Datei parsen

			REPEAT

				brwcsncpy( ADR(_GetCsvDat.utfCsvString), _plLineAdress[_wStartLine], MIN(299, _pwLineLen[_wStartLine]));
				_GetCsvDat();
				_wStartLine := _wStartLine + 1;

				IF _GetCsvDat.RowType = 200 AND _GetCsvDat.csvTextRow.LCID = _wActLCID AND _wIdxParamTxt <= MNTXT_MAX_IDX_TXT_PARAMETER THEN

					_TxtLine.wNumber := _GetCsvDat.csvTextRow.TextNo;
					_TxtLine.wFunctionID := _GetCsvDat.csvTextRow.FunctionID;
					_TxtLine.utfText := _GetCsvDat.csvTextRow.utfText;

					_dowParTxt(enable := TRUE, ident := _CheckDoPar.doId, Offset := SIZEOF(_TxtLine)*_wIdxParamTxt, pSource := ADR(_TxtLine), len := SIZEOF(_TxtLine));

					_wIdxParamTxt := _wIdxParamTxt + 1;

				ELSIF _GetCsvDat.RowType = 210 AND _GetCsvDat.csvHelpTextRow.LCID = _wActLCID AND _wIdxParamHelpTxt <= MNTXT_MAX_IDX_TXT_PARAMETER AND MNTXT_LOAD_PARAMTERHELPTEXT THEN

					_TxtHelpLine.wNumber := _GetCsvDat.csvHelpTextRow.TextNo;
					_TxtHelpLine.wFunctionID := _GetCsvDat.csvHelpTextRow.FunctionID;

					// _TxtHelpLine.utfText := _GetCsvDat.csvHelpTextRow.utfHelpText;

					_utfRC(pInput := ADR(_GetCsvDat.csvHelpTextRow.utfHelpText), pOutput := ADR(_TxtHelpLine.utfText), lSizeOutput := SIZEOF(_TxtHelpLine.utfText), xWSTRING := TRUE);

					_dowParHlpTxt(enable := TRUE, ident := _CheckDoParHlp.doId, Offset := SIZEOF(_TxtHelpLine)*_wIdxParamHelpTxt, pSource := ADR(_TxtHelpLine), len := SIZEOF(_TxtHelpLine));

					_wIdxParamHelpTxt := _wIdxParamHelpTxt + 1;

				END_IF

				_lCycleCounter := _lCycleCounter + 1;

				UNTIL

				_lCycleCounter > 20 OR (_wIdxParamTxt > MNTXT_MAX_IDX_TXT_PARAMETER AND _wIdxParamHelpTxt > MNTXT_MAX_IDX_TXT_PARAMETER) OR _wStartLine > _CountLines.CntLines

			END_REPEAT

			IF (_wIdxParamTxt > MNTXT_MAX_IDX_TXT_PARAMETER AND _wIdxParamHelpTxt > MNTXT_MAX_IDX_TXT_PARAMETER) OR _wStartLine > _CountLines.CntLines THEN

				IFmnTxt.Out.wCntParamTxt := _wIdxParamTxt;
				IFmnTxt.Out.wCntParamHlpTxt := _wIdxParamHelpTxt;
				_LoadState := _ls_load_paramtxt_08;

			END_IF

		_ls_load_paramtxt_08:

			// Speicher frei geben

			_MemPartFree(enable := TRUE, ident := _MemPartCreate.ident, mem := _lAdrFile);

			IF _MemPartFree.status = ERR_OK THEN

				_LoadState := _ls_idle;
				IFmnTxt.Out.wSelectLanguageStatus := MNTXT_STAT_OK;

			ELSIF _MemPartFree.status <> ERR_FUB_BUSY THEN

				IFmnTxt.Out.wSelectLanguageStatus := MNTXT_STAT_ERRPARAMTXT;
				_LoadState := _ls_error;

			END_IF

		_ls_error:

			// Fehlerzustand

	END_CASE

END_PROGRAM
```

#### mnTxtInit.st - Initialization code
```iecst
(********************************************************************
 * COPYRIGHT -- Herbert Kannegiesser GmbH
 ********************************************************************
 * Program: mnTxt
 * File: mnTxtInit.st
 * Author: hunholz
 * Created: November 25, 2011
 ********************************************************************
 * Implementation of program mnTxt
 ********************************************************************)

PROGRAM _INIT

	// Packet-Version auslesen mit MO_ver aus SYS_lib und für den Additional Status zur Verfügung stellen

	_sPkgName := 'mnTxt';

	IF ( MO_ver(ADR(_sPkgName), 0, ADR(_VerStruc)) = 0 ) THEN

		brsmemcpy(ADR(mnTxtStatAd.sPkgVersion), ADR(_VerStruc.version), SIZEOF(_VerStruc.version));

	ELSE

		mnTxtStatAd.sPkgVersion := '---';

	END_IF

	brsmemset(ADR(IFmnTxt.Out), 0, SIZEOF(IFmnTxt.Out));

	IFmnTxt.Out.wSelectLanguageStatus := MNTXT_STAT_INIT;

	REPEAT

		//===================================
		// Speicher zum Parsen bereitstellen
		//===================================

		// Bedarf berechnen

		_lLineMem := (((SIZEOF(_plLineAdress) + SIZEOF(_pwLineLen)) / 8) + 2 ) * 8;

		_lLineMem := _lLineMem + ((MNTXT_TEMPREADCSVSIZE / 8) + 2) * 8;

		_lLineMem := _lLineMem + 1000;

		_MemPartCreate(enable := TRUE, len := _lLineMem);

		IF _MemPartCreate.status <> ERR_OK THEN

			IFmnTxt.Out.wSelectLanguageStatus := MNTXT_STAT_ERRMEM;
			EXIT;

		END_IF

		// Zeilenadresstabelle
		_MemPartAlloc(enable := TRUE, ident := _MemPartCreate.ident, len := SIZEOF(_plLineAdress) + SIZEOF(_pwLineLen) );

		IF _MemPartAlloc.status <> ERR_OK THEN

			IFmnTxt.Out.wSelectLanguageStatus := MNTXT_STAT_ERRMEM;
			EXIT;

		END_IF

		_lAdrLineAdress := _MemPartAlloc.mem;
		_plLineAdress ACCESS _lAdrLineAdress;

		_lAdrLineLen := _lAdrLineAdress + SIZEOF(_plLineAdress);
		_pwLineLen ACCESS _lAdrLineLen;

		//LCID_Tabelle einlesen

		_FileInfo(enable := TRUE, pDevice := ADR(KG_DEVICE_COMPACTFLASH), pName := ADR('Language\lcid.csv'), pInfo := ADR(_fiFileInfo));

		IF _FileInfo.status <> ERR_OK THEN

			IFmnTxt.Out.wSelectLanguageStatus := MNTXT_STAT_ERRLCID;
			EXIT;

		END_IF

		_MemPartAlloc(enable := TRUE, ident := _MemPartCreate.ident, len := _fiFileInfo.size-SIZEOF(KGBOM) );

		IF _MemPartAlloc.status <> ERR_OK THEN

			IFmnTxt.Out.wSelectLanguageStatus := MNTXT_STAT_ERRMEM;
			EXIT;

		END_IF

		_lAdrFile := _MemPartAlloc.mem;

		_FileOpen(enable := TRUE, pDevice := ADR(KG_DEVICE_COMPACTFLASH), pFile := ADR('Language\lcid.csv'), mode := fiREAD_ONLY);

		IF _FileOpen.status <> ERR_OK THEN

			IFmnTxt.Out.wSelectLanguageStatus := MNTXT_STAT_ERRLCID;
			EXIT;

		END_IF

		_FileRead(enable := TRUE, ident := _FileOpen.ident, offset := SIZEOF(KGBOM),pDest := _lAdrFile, len :=  _fiFileInfo.size-SIZEOF(KGBOM) ) ;

		_FileClose(enable := TRUE, ident := _FileOpen.ident);

		IF _FileRead.status <> ERR_OK THEN

			IFmnTxt.Out.wSelectLanguageStatus := MNTXT_STAT_ERRLCID;
			EXIT;

		END_IF

		// Zeilen in der Datei zählen und Startadressen ermitteln

		_CountLines.enable := TRUE;
		_CountLines.pFile := _lAdrFile;
		_CountLines.FileSize := _fiFileInfo.size - SIZEOF(KGBOM);
		_CountLines.MaxLines := MNTXT_MAXPARSELINES;
		_CountLines.pAdresses := _lAdrLineAdress;
		_CountLines.pLens := _lAdrLineLen;

		_CountLines();

		IF _CountLines.status <> ERR_OK THEN

			IFmnTxt.Out.wSelectLanguageStatus := MNTXT_STAT_ERRLCID;
			EXIT;

		END_IF

		// Zeilen auslesen und LCID-Werte ermitteln

		_xGermanExist := FALSE;
		_wStartLine := 1;
		_wIdxLCID := 0;
		_GetCsvDat.enable := TRUE;

		REPEAT

			brwcsncpy( ADR(_GetCsvDat.utfCsvString), _plLineAdress[_wStartLine], MIN(299, _pwLineLen[_wStartLine]));
			_GetCsvDat();
			_wStartLine := _wStartLine + 1;

			IF _GetCsvDat.RowType = 248 AND _GetCsvDat.CsvLCIDrow.LCID > 0 THEN

				IFmnTxt.Out.wLCIDs[_wIdxLCID] := _GetCsvDat.CsvLCIDrow.LCID;
				_wIdxLCID := _wIdxLCID + 1;

				IF _GetCsvDat.CsvLCIDrow.LCID = MNTXT_LCID_GERMAN THEN
					_xGermanExist := TRUE;
				END_IF

			END_IF

			UNTIL
			_wIdxLCID > MNTXT_MAX_IDX_LCID OR _wStartLine > _CountLines.CntLines
		END_REPEAT

		IFmnTxt.Out.wCntLCID := _wIdxLCID;

		_MemPartFree(enable := TRUE, ident := _MemPartCreate.ident, mem := _lAdrFile);

		IF IFmnTxt.Out.wCntLCID = 0 THEN

			IFmnTxt.Out.wSelectLanguageStatus := MNTXT_STAT_ERRLCID;
			EXIT;

		END_IF

		//##############################################################################

		IFmnTxt.Out.wSelectLanguageStatus := MNTXT_STAT_NOLANGUAGE;

		_initState := _is_checkFunctionTxt;
		_xInitOK := FALSE;
		_xInitDone := FALSE;

		UNTIL
		TRUE
	END_REPEAT

	REPEAT

		CASE _initState OF

			// Datenobjekte für Funktionstexte prüfen und ggf. anlegen
			_is_checkFunctionTxt:

				IFmnTxt.Out.ptrFunctionTxtList := 0;
				IFmnTxt.Out.wCntFunctionTxt := 0;

				_lLenFuncTxt := SIZEOF(_TxtLine)*(MNTXT_MAX_IDX_TXT_FUNCTION+1);

				IF MNTXT_LOAD_FUNCTIONTEXT THEN

					_CheckDoFunc(Enable := TRUE, pName := ADR(MNTXT_DATOBJNAME_FUNTXT), MinLen := _lLenFuncTxt, NomLen := _lLenFuncTxt, Create := TRUE, MemType := doUSRROM);

					IF _CheckDoFunc.Status <> ERR_FUB_BUSY THEN

						// DO mit Templatetexten füllen, wenn es neu angelegt wurde

						IF _CheckDoFunc.Status = KG_INFO_DO_NEW OR _CheckDoFunc.Status = ERR_OK THEN

							_debFunctionTxtList ACCESS _CheckDoFunc.doMem;

							IFmnTxt.Out.ptrFunctionTxtList := _CheckDoFunc.doMem;

							IF _CheckDoFunc.Status = KG_INFO_DO_NEW THEN

								_initState := _is_writeFunctionTxt;
								_ii := 0;

							ELSE

								_initState := _is_checkInstanceTxt;

							END_IF

						ELSE

							_xInitDone := TRUE;
							IFmnTxt.Out.wSelectLanguageStatus := _CheckDoFunc.Status;

						END_IF

					END_IF

				ELSE

					_initState := _is_checkInstanceTxt;

				END_IF

			_is_writeFunctionTxt:

				REPEAT

					_TxtLine.wNumber 		:= _ii;
					_TxtLine.wFunctionID 	:= _ii;
					_TxtLine.utfText		:= "Function";
					_utfNo					:= UINT_TO_WSTRING(_ii);
					brwcscat(ADR(_TxtLine.utfText), ADR(_utfNo));

					_dowFuncTxt(enable := TRUE, ident := _CheckDoFunc.doId, Offset := SIZEOF(_TxtLine)*_ii, pSource := ADR(_TxtLine), len := SIZEOF(_TxtLine));

					IF _dowFuncTxt.status <> ERR_OK THEN

						IFmnTxt.Out.wSelectLanguageStatus := MNTXT_STAT_ERRDATOBJ;
						_xInitDone := TRUE;
						EXIT;

					END_IF

					_ii := _ii + 1;

					UNTIL
					((_ii MOD 10) = 0) OR _ii > MNTXT_MAX_IDX_TXT_FUNCTION
				END_REPEAT

				IF _ii > MNTXT_MAX_IDX_TXT_FUNCTION THEN

					_initState := _is_checkInstanceTxt;

				END_IF

			// Datenobjekte für Instanztexte prüfen und ggf. anlegen
			_is_checkInstanceTxt:

				IFmnTxt.Out.ptrInstanceTxtList := 0;
				IFmnTxt.Out.wCntInstanceTxt		:= 0;

				_lLenInstTxt := SIZEOF(_TxtLine)*(MNTXT_MAX_IDX_TXT_INSTANCE + 1);

				IF MNTXT_LOAD_INSTANCETEXT THEN

					_CheckDoInst(Enable := TRUE, pName := ADR(MNTXT_DATOBJNAME_INSTXT), MinLen := _lLenInstTxt, NomLen := _lLenInstTxt, Create := TRUE, MemType := doUSRROM);

					IF _CheckDoInst.Status <> ERR_FUB_BUSY THEN

						// DO mit Templatetexten füllen, wenn es neu angelegt wurde

						IF _CheckDoInst.Status = KG_INFO_DO_NEW OR _CheckDoInst.Status = ERR_OK THEN

							IFmnTxt.Out.ptrInstanceTxtList := _CheckDoInst.doMem;

							_debInstanceTxtList ACCESS _CheckDoInst.doMem;

							IF _CheckDoInst.Status = KG_INFO_DO_NEW THEN

								_ii := 0;
								_initState := _is_writeInstanceTxt;

							ELSE

								_initState := _is_checkParTxt;

							END_IF

						ELSE

							IFmnTxt.Out.wSelectLanguageStatus := _CheckDoInst.Status;
							_xInitDone := TRUE;

						END_IF

					END_IF

				ELSE

					_initState := _is_checkParTxt;

				END_IF

			_is_writeInstanceTxt:

				REPEAT

					_TxtLine.wNumber 		:= _ii;
					_TxtLine.wFunctionID 	:= _ii;
					_TxtLine.utfText		:= "Instance";
					_utfNo					:= UINT_TO_WSTRING(_ii);
					brwcscat(ADR(_TxtLine.utfText), ADR(_utfNo));

					_dowInstTxt(enable := TRUE, ident := _CheckDoInst.doId, Offset := SIZEOF(_TxtLine)*_ii, pSource := ADR(_TxtLine), len := SIZEOF(_TxtLine));

					IF _dowInstTxt.status <> ERR_OK THEN

						IFmnTxt.Out.wSelectLanguageStatus := MNTXT_STAT_ERRDATOBJ;
						_xInitDone := TRUE;
						EXIT;

					END_IF

					_ii := _ii + 1;

					UNTIL
					((_ii MOD 10) = 0) OR _ii > MNTXT_MAX_IDX_TXT_INSTANCE
				END_REPEAT

				IF _ii > MNTXT_MAX_IDX_TXT_INSTANCE THEN

					_initState := _is_checkParTxt;

				END_IF

			// Datenobjekte für Parametertexte prüfen und ggf. anlegen
			_is_checkParTxt:

				IFmnTxt.Out.ptrParamTxtList := 0;
				IFmnTxt.Out.wCntParamTxt := 0;

				_lLenParTxt := SIZEOF(_TxtLine)*(MNTXT_MAX_IDX_TXT_PARAMETER + 1);

				IF MNTXT_LOAD_PARAMETERTEXT THEN

					_CheckDoPar(Enable := TRUE, pName := ADR(MNTXT_DATOBJNAME_PARTXT), MinLen := _lLenParTxt, NomLen := _lLenParTxt, Create := TRUE, MemType := doUSRROM);

					IF _CheckDoPar.Status <> ERR_FUB_BUSY THEN

						// DO mit Templatetexten füllen, wenn es neu angelegt wurde

						IF _CheckDoPar.Status = KG_INFO_DO_NEW OR _CheckDoPar.Status = ERR_OK THEN

							_debParameterTxtList ACCESS _CheckDoPar.doMem;

							IFmnTxt.Out.ptrParamTxtList := _CheckDoPar.doMem;

							IF _CheckDoPar.Status = KG_INFO_DO_NEW THEN

								_ii := 0;
								_initState := _is_writeParTxt;

							ELSE

								_initState := _is_checkParHlpTxt;

							END_IF

						ELSE

							IFmnTxt.Out.wSelectLanguageStatus := _CheckDoPar.Status;
							_xInitDone := TRUE;

						END_IF

					END_IF

				ELSE

					_initState := _is_checkParHlpTxt;

				END_IF

			_is_writeParTxt:

				REPEAT

					_TxtLine.wNumber 		:= _ii;
					_TxtLine.wFunctionID 	:= _ii;
					_TxtLine.utfText		:= "Parameter";
					_utfNo					:= UINT_TO_WSTRING(_ii);
					brwcscat(ADR(_TxtLine.utfText), ADR(_utfNo));

					_dowParTxt(enable := TRUE, ident := _CheckDoPar.doId, Offset := SIZEOF(_TxtLine)*_ii, pSource := ADR(_TxtLine), len := SIZEOF(_TxtLine));

					IF _dowParTxt.status <> ERR_OK THEN

						IFmnTxt.Out.wSelectLanguageStatus := MNTXT_STAT_ERRDATOBJ;
						_xInitDone := TRUE;
						EXIT;

					END_IF

					_ii := _ii + 1;

					UNTIL
					((_ii MOD 10) = 0) OR _ii > MNTXT_MAX_IDX_TXT_PARAMETER
				END_REPEAT

				IF _ii > MNTXT_MAX_IDX_TXT_PARAMETER THEN

					_initState := _is_checkParHlpTxt;

				END_IF

			// Datenobjekte für Parameterhilfstexte prüfen und ggf. anlegen
			_is_checkParHlpTxt:

				IFmnTxt.Out.ptrParamHelpTxtList := 0;
				IFmnTxt.Out.wCntParamHlpTxt := 0;

				_lLenParHlpTxt := SIZEOF(_TxtHelpLine)*(MNTXT_MAX_IDX_TXT_PARAMETER + 1);

				IF MNTXT_LOAD_PARAMTERHELPTEXT THEN

					_CheckDoParHlp(Enable := TRUE, pName := ADR(MNTXT_DATOBJNAME_PARHELPTXT), MinLen := _lLenParHlpTxt, NomLen := _lLenParHlpTxt, Create := TRUE, MemType := doUSRROM);

					IF _CheckDoParHlp.Status <> ERR_FUB_BUSY THEN

						// DO mit Templatetexten füllen, wenn es neu angelegt wurde

						IF _CheckDoParHlp.Status = KG_INFO_DO_NEW OR _CheckDoParHlp.Status = ERR_OK THEN

							_debParameterHlpTxtList ACCESS _CheckDoParHlp.doMem;

							IFmnTxt.Out.ptrParamHelpTxtList := _CheckDoParHlp.doMem;

							IF _CheckDoParHlp.Status = KG_INFO_DO_NEW THEN

								_ii := 0;
								_initState := _is_writeParHlpTxt;

							ELSE

								_initState := _is_checkMsgCnt;

							END_IF

						ELSE

							IFmnTxt.Out.wSelectLanguageStatus := _CheckDoParHlp.Status;
							_xInitDone := TRUE;

						END_IF

					END_IF

				ELSE

					_initState := _is_checkMsgCnt;

				END_IF

			_is_writeParHlpTxt:

				REPEAT

					_TxtHelpLine.wNumber 		:= _ii;
					_TxtHelpLine.wFunctionID 	:= _ii;
					_TxtHelpLine.utfText		:= "Parameter Help";
					_utfNo						:= UINT_TO_WSTRING(_ii);
					brwcscat(ADR(_TxtHelpLine.utfText), ADR(_utfNo));

					_dowParHlpTxt(enable := TRUE, ident := _CheckDoParHlp.doId, Offset := SIZEOF(_TxtHelpLine)*_ii, pSource := ADR(_TxtHelpLine), len := SIZEOF(_TxtHelpLine));

					IF _dowParHlpTxt.status <> ERR_OK THEN

						IFmnTxt.Out.wSelectLanguageStatus := MNTXT_STAT_ERRDATOBJ;
						_xInitDone := TRUE;
						EXIT;

					END_IF

					_ii := _ii + 1;

					UNTIL
					((_ii MOD 10) =0) OR _ii > MNTXT_MAX_IDX_TXT_PARAMETER
				END_REPEAT

				IF _ii > MNTXT_MAX_IDX_TXT_PARAMETER THEN

					_initState := _is_checkMsgCnt;

				END_IF

			// Anzahl Meldungen ermitteln
			_is_checkMsgCnt:

				REPEAT

					_doiMsgCfg(enable := TRUE, pName := ADR('CfgMsgStat'));

					IF _doiMsgCfg.status <> ERR_OK THEN

						IFmnTxt.Out.wSelectLanguageStatus := MNTXT_STAT_ERRMSGCFG;
						_xInitDone := TRUE;
						EXIT;

					END_IF

					IF _doiMsgCfg.len < 2 THEN

						IFmnTxt.Out.wSelectLanguageStatus := MNTXT_STAT_ERRMSGCFG;
						_xInitDone := TRUE;
						EXIT;

					END_IF

					_MsgCfgList ACCESS _doiMsgCfg.pDatObjMem + 2;

					_lLenMsg := (_doiMsgCfg.len-2) / SIZEOF(_MsgCfgList[0]);

					_initState := _is_checkMsgTxt;

					UNTIL
					TRUE

				END_REPEAT

			// Datenobjekte für Meldungstexte prüfen und ggf. anlegen
			_is_checkMsgTxt:

				// Referenz auf die Meldungskonfiguration holen und Anzahl der möglichen Meldungen
				// ermitteln

				IFmnTxt.Out.ptrMessageTxtList := 0;
				IFmnTxt.Out.wCntMessageTxt := 0;

				_lLenMsgTxt := SIZEOF(_TxtLine)* _lLenMsg;

				_CheckDoMsg(Enable := TRUE, pName := ADR(MNTXT_DATOBJNAME_MSGTXT), MinLen := _lLenMsgTxt, NomLen := _lLenMsgTxt, Create := TRUE, MemType := doUSRROM);

				IF _CheckDoMsg.Status <> ERR_FUB_BUSY THEN

					// DO mit Templatetexten füllen, wenn es neu angelegt wurde
					IF _CheckDoMsg.Status = KG_INFO_DO_NEW OR _CheckDoMsg.Status = ERR_OK THEN

						_debMessageTxtList ACCESS _CheckDoMsg.doMem;

						IFmnTxt.Out.ptrMessageTxtList := _CheckDoMsg.doMem;
						IFmnTxt.Out.wCntMessageTxt := UDINT_TO_UINT(_lLenMsg);

						_ii := 0;

						_initState := _is_writeMsgTxt;

					ELSE

						IFmnTxt.Out.wSelectLanguageStatus := _CheckDoMsg.Status;
						_xInitDone := TRUE;

					END_IF

				END_IF

			_is_writeMsgTxt:

				IF _CheckDoMsg.Status = KG_INFO_DO_NEW AND _lLenMsg > 0 THEN

					REPEAT

						_TxtLine.wNumber 		:= _MsgCfgList[_ii].wMsgNumber;
						_TxtLine.wFunctionID 	:= _MsgCfgList[_ii].wFunction_ID;
						_TxtLine.wInstance		:= _MsgCfgList[_ii].wInstance;
						_TxtLine.utfText		:= "Message";
						_utfNo					:= UINT_TO_WSTRING(_MsgCfgList[_ii].wMsgNumber);
						brwcscat(ADR(_TxtLine.utfText), ADR(_utfNo));

						_dowMsgTxt(enable := TRUE, ident := _CheckDoMsg.doId, Offset := SIZEOF(_TxtLine)*_ii, pSource := ADR(_TxtLine), len := SIZEOF(_TxtLine));

						IF _dowMsgTxt.status <> ERR_OK THEN

							IFmnTxt.Out.wSelectLanguageStatus := MNTXT_STAT_ERRDATOBJ;
							_xInitDone := TRUE;
							EXIT;

						END_IF

						_ii := _ii + 1;

						UNTIL
						((_ii MOD 10) = 0) OR _ii >= _lLenMsg

					END_REPEAT

					IF _ii >= _lLenMsg THEN

						_initState := _is_checkMsgHlpTxt;

					END_IF

				ELSE

					_initState := _is_checkMsgHlpTxt;

				END_IF

			// Datenobjekte für Meldungstexte prüfen und ggf. anlegen
			_is_checkMsgHlpTxt:

				IFmnTxt.Out.ptrMessageHelpTxtList := 0;
				IFmnTxt.Out.wCntMessageHlpTxt := 0;

				_lLenMsgHlpTxt := SIZEOF(_TxtHelpLine)* _lLenMsg;

				_CheckDoMsgHlp(Enable := TRUE, pName := ADR(MNTXT_DATOBJNAME_MSGHELPTXT), MinLen := _lLenMsgHlpTxt, NomLen := _lLenMsgHlpTxt, Create := TRUE, MemType := doUSRROM);

				IF _CheckDoMsgHlp.Status <> ERR_FUB_BUSY THEN

					// DO mit Templatetexten füllen, wenn es neu angelegt wurde
					IF _CheckDoMsgHlp.Status = KG_INFO_DO_NEW OR _CheckDoMsgHlp.Status = ERR_OK THEN

						_debMessageHlpTxtList ACCESS _CheckDoMsgHlp.doMem;

						IFmnTxt.Out.ptrMessageHelpTxtList := _CheckDoMsgHlp.doMem;
						IFmnTxt.Out.wCntMessageHlpTxt := UDINT_TO_UINT(_lLenMsg);

						_ii := 0;

						_initState := _is_writeMsgHlpTxt;

					ELSE

						IFmnTxt.Out.wSelectLanguageStatus := _CheckDoMsg.Status;
						_xInitDone := TRUE;

					END_IF

				END_IF

			_is_writeMsgHlpTxt:

				IF _CheckDoMsgHlp.Status = KG_INFO_DO_NEW AND _lLenMsg > 0 THEN

					REPEAT

						_TxtHelpLine.wNumber 		:= _MsgCfgList[_ii].wMsgNumber;
						_TxtHelpLine.wFunctionID 	:= _MsgCfgList[_ii].wFunction_ID;
						_TxtHelpLine.wInstance		:= _MsgCfgList[_ii].wInstance;
						_TxtHelpLine.utfText		:= "Message Help";
						_utfNo					:= UINT_TO_WSTRING(_MsgCfgList[_ii].wMsgNumber);
						brwcscat(ADR(_TxtHelpLine.utfText), ADR(_utfNo));

						_dowMsgHlpTxt(enable := TRUE, ident := _CheckDoMsgHlp.doId, Offset := SIZEOF(_TxtHelpLine)*_ii, pSource := ADR(_TxtHelpLine), len := SIZEOF(_TxtHelpLine));

						IF _dowMsgHlpTxt.status <> ERR_OK THEN

							IFmnTxt.Out.wSelectLanguageStatus := MNTXT_STAT_ERRDATOBJ;
							_xInitDone := TRUE;
							EXIT;

						END_IF

						_ii := _ii + 1;

						UNTIL
						((_ii MOD 10)) = 0 OR	_ii >= _lLenMsg
					END_REPEAT

					IF _ii >= _lLenMsg THEN
						_xInitDone := TRUE;
						_xInitOK := TRUE;
					END_IF

				ELSE

					_xInitDone := TRUE;
					_xInitOK := TRUE;

				END_IF

		END_CASE

		UNTIL
		_xInitDone
	END_REPEAT

	mnTxtPar;

END_PROGRAM
```

#### mnTxt.typ - Local data types
```iecst
(********************************************************************
 * COPYRIGHT -- Herbert Kannegiesser GmbH
 ********************************************************************
 * Program: mnTxt
 * File: mnTxt.typ
 * Author: hunholz
 * Created: November 25, 2011
 ********************************************************************
 * Local data types of program mnTxt
 ********************************************************************)

TYPE
	_mntxt_loadstate_enum :
		(
		_ls_idle := 0,
		_ls_load_functiontxt_01 := 100,
		_ls_load_functiontxt_02,
		_ls_load_functiontxt_03,
		_ls_load_functiontxt_04,
		_ls_load_functiontxt_05,
		_ls_load_functiontxt_06,
		_ls_load_functiontxt_07,
		_ls_load_functiontxt_08,
		_ls_load_instancetxt_01 := 200,
		_ls_load_instancetxt_02,
		_ls_load_instancetxt_03,
		_ls_load_instancetxt_04,
		_ls_load_instancetxt_05,
		_ls_load_instancetxt_06,
		_ls_load_instancetxt_07,
		_ls_load_instancetxt_08,
		_ls_load_messagetxt_01 := 300,
		_ls_load_messagetxt_02,
		_ls_load_messagetxt_03,
		_ls_load_messagetxt_04,
		_ls_load_messagetxt_05,
		_ls_load_messagetxt_06,
		_ls_load_messagetxt_07,
		_ls_load_messagetxt_08,
		_ls_load_paramtxt_01 := 400,
		_ls_load_paramtxt_02,
		_ls_load_paramtxt_03,
		_ls_load_paramtxt_04,
		_ls_load_paramtxt_05,
		_ls_load_paramtxt_06,
		_ls_load_paramtxt_07,
		_ls_load_paramtxt_08,
		_ls_error := 65535
		);
	_mntxt_initstate_enum :
		(
		_is_checkFunctionTxt,
		_is_writeFunctionTxt,
		_is_checkInstanceTxt,
		_is_writeInstanceTxt,
		_is_checkParTxt,
		_is_writeParTxt,
		_is_checkParHlpTxt,
		_is_writeParHlpTxt,
		_is_checkMsgCnt,
		_is_checkMsgTxt,
		_is_writeMsgTxt,
		_is_checkMsgHlpTxt,
		_is_writeMsgHlpTxt
		);
	_mntxt_rem_typ : 	STRUCT
		dtFuncTxt : DATE_AND_TIME;
		dtInstTxt : DATE_AND_TIME;
		dtParTxt : DATE_AND_TIME;
		dtMsgTxt : DATE_AND_TIME;
	END_STRUCT;
END_TYPE
```

#### mnTxt.var - Local variables
```iecst
(********************************************************************
 * COPYRIGHT -- Herbert Kannegiesser GmbH
 ********************************************************************
 * Program: mnTxt
 * File: mnTxt.var
 * Author: hunholz
 * Created: November 25, 2011
 ********************************************************************
 * Local variables of program mnTxt
 ********************************************************************)
(*Hilfsvariablen*)
VAR
	_ii : UINT;
	_utfNo : WSTRING[5];
	_TxtLine : mnTxt_TxtLine_Typ;
	_TxtHelpLine : mnTxt_HelpTxtLine_Typ;
END_VAR
(*Function-Txt Datenobjekt prüfen, anlegen, füllen*)
VAR
	_dowFuncTxt : DatObjWrite;
	_debFunctionTxtList : REFERENCE TO ARRAY[0..MNTXT_MAX_IDX_TXT_FUNCTION] OF mnTxt_TxtLine_Typ;
	_lLenFuncTxt : UDINT;
END_VAR
(*Instance-Txt Datenobjekt prüfen, anlegen, füllen*)
VAR
	_dowInstTxt : DatObjWrite;
	_debInstanceTxtList : REFERENCE TO ARRAY[0..MNTXT_MAX_IDX_TXT_INSTANCE] OF mnTxt_TxtLine_Typ;
	_lLenInstTxt : UDINT;
END_VAR
(*Parameter-Txt Datenobjekt prüfen, anlegen, füllen*)
VAR
	_dowParTxt : DatObjWrite;
	_debParameterTxtList : REFERENCE TO ARRAY[0..MNTXT_MAX_IDX_TXT_PARAMETER] OF mnTxt_TxtLine_Typ;
	_lLenParTxt : UDINT;
END_VAR
(*Parameter-HlpTxt Datenobjekt prüfen, anlegen, füllen*)
VAR
	_dowParHlpTxt : DatObjWrite;
	_debParameterHlpTxtList : REFERENCE TO ARRAY[0..MNTXT_MAX_IDX_TXT_PARAMETER] OF mnTxt_HelpTxtLine_Typ;
	_lLenParHlpTxt : UDINT;
END_VAR
(*Meldungs-Txt Datenobjekt prüfen, anlegen, füllen*)
VAR
	_dowMsgTxt : DatObjWrite;
	_debMessageTxtList : REFERENCE TO ARRAY[0..65535] OF mnTxt_TxtLine_Typ;
	_lLenMsgTxt : UDINT;
END_VAR
(*Meldungs-HlpTxt Datenobjekt prüfen, anlegen, füllen*)
VAR
	_dowMsgHlpTxt : DatObjWrite;
	_debMessageHlpTxtList : REFERENCE TO ARRAY[0..65535] OF mnTxt_HelpTxtLine_Typ;
	_lLenMsgHlpTxt : UDINT;
	_doiMsgCfg : DatObjInfo;
	_lLenMsg : UDINT;
	_MsgCfgList : REFERENCE TO ARRAY[0..65535] OF MsgCfgLine_Typ;
	_LoadState : _mntxt_loadstate_enum;
END_VAR
VAR CONSTANT
	_MemPartCreate : AsMemPartCreate := (0);
END_VAR
VAR
	_MemPartAlloc : AsMemPartAlloc;
	_plLineAdress : REFERENCE TO ARRAY[1..MNTXT_MAXPARSELINES] OF UDINT;
	_pwLineLen : REFERENCE TO ARRAY[1..MNTXT_MAXPARSELINES] OF UINT;
	_fiFileInfo : fiFILE_INFO;
	_FileInfo : FileInfo;
	_FileOpen : FileOpen;
	_lAdrFile : UDINT;
	_FileRead : FileRead;
	_FileClose : FileClose;
	_CountLines : mnParam_CountLines;
	_lAdrLineAdress : UDINT;
	_lAdrLineLen : UDINT;
	_wStartLine : UINT;
	_wIdxLCID : UINT;
	_GetCsvDat : mnParam_GetCsvDat;
	_MemPartFree : AsMemPartFree;
END_VAR
VAR RETAIN
	_wActLCID : UINT;
END_VAR
VAR
	_xGermanExist : BOOL;
	_lCycleCounter : UDINT;
	_wIdxFunctionTxt : UINT;
	_wIdxInstanceTxt : UINT;
	_wIdxMessageTxt : UINT;
	_wIdxMessageHelpTxt : UINT;
	_wIdxParamTxt : UINT;
	_wIdxParamHelpTxt : UINT;
	_sPkgName : STRING[11];
	_VerStruc : MoVerStruc_typ;
	_lLineMem : UDINT;
	_xInitOK : BOOL;
	_initState : _mntxt_initstate_enum;
	_CheckDoFunc : kgCheckDo;
	_CheckDoInst : kgCheckDo;
	_xInitDone : BOOL;
	_CheckDoPar : kgCheckDo;
	_CheckDoParHlp : kgCheckDo;
	_CheckDoMsg : kgCheckDo;
	_CheckDoMsgHlp : kgCheckDo;
	_utfRC : _utfReplaceCtrl;
	_sLCID : STRING[7];
	_sPath : STRING[256];
END_VAR
```

#### _utfReplaceCtrl.st - Replace Linefeed
```iecst
(********************************************************************
 * COPYRIGHT -- Herbert Kannegiesser GmbH
 ********************************************************************
 * Program: mnTxt
 * File: _utfReplaceCtrl.st
 * Author: hunholz
 * Created: June 22, 2012
 ********************************************************************
 * Implementation of program mnTxt
 ********************************************************************)

(* Replace Linefeed *)
FUNCTION_BLOCK _utfReplaceCtrl

	wStatus := ERR_OK;

	IF pInput = 0 OR pOutput = 0 THEN
		wStatus := KG_ERR_NULPOINTER;
		RETURN;
	END_IF

	IF xWSTRING THEN

		IF lSizeOutput < 2 THEN

			wStatus := KG_ERR_WRONGSIZES;
			RETURN;

		END_IF

		_utfInput ACCESS pInput;

		IF (brwcslen(pInput) * 2) + 2 > MIN(lSizeOutput,2048) THEN

			brsmemcpy(pOutput,pInput,MIN(lSizeOutput,2048));
			_wChar1 ACCESS pOutput + (MIN(lSizeOutput,2048)-2);
			_wChar1 := 0;

		ELSE

			brwcscpy(pOutput, pInput);

		END_IF

		_utfOutput ACCESS pOutput;

		_pOutput := pOutput;

		REPEAT

			_lChar1 := brwcschr(_pOutput, 16#5C);
			_lChar2 := brwcschr(_pOutput, 16#6E);

			IF _lChar1 > 0 AND _lChar2 > 0 AND (_lChar1+2) = _lChar2 THEN

				_wChar1 ACCESS _lChar1;
				_wChar2 ACCESS _lChar2;

				_wChar1 := 16#0D;
				_wChar2 := 16#0A;

			ELSIF _lChar1 > 0 AND _lChar2 > 0 THEN

				IF _lChar1 < _lChar2 THEN
					_pOutput := _lChar1 + 2;
				ELSE
					_pOutput := _lChar2 + 2;
				END_IF

			END_IF

			UNTIL
			_lChar1 = 0 OR _lChar2 = 0
		END_REPEAT

	ELSE

		IF lSizeOutput = 0 THEN

			wStatus := KG_ERR_WRONGSIZES;
			RETURN;

		END_IF

		_sInput ACCESS pInput;

		_sOutput ACCESS pOutput;

		IF INT_TO_UDINT(LEN(_sInput) + 1)	> MIN(lSizeOutput,256) THEN

			brsmemcpy(pOutput,pInput,MIN(lSizeOutput,256));
			_bChar1 ACCESS pOutput + (MIN(lSizeOutput,256)-1);
			_bChar1 := 0;

		ELSE

			_sOutput := _sInput;

		END_IF

		REPEAT

			_iPos := FIND(_sOutput,'\n');

			IF _iPos > 0 THEN

				_sOutput := REPLACE(_sOutput, '$R$N', 2, _iPos);

			END_IF

			UNTIL
			_iPos = 0
		END_REPEAT

	END_IF

END_FUNCTION_BLOCK
```

#### mnTxt.fun
```iecst
(********************************************************************
 * COPYRIGHT -- Herbert Kannegiesser GmbH
 ********************************************************************
 * Program: mnTxt
 * File: mnTxt.fun
 * Author: hunholz
 * Created: June 22, 2012
 ********************************************************************
 * Functions and function blocks of program mnTxt
 ********************************************************************)

FUNCTION_BLOCK _utfReplaceCtrl (*Replace Linefeed*)
	VAR_INPUT
		pInput : UDINT;
		pOutput : UDINT;
		lSizeOutput : UDINT;
		xWSTRING : BOOL;
	END_VAR
	VAR_OUTPUT
		wStatus : UINT;
	END_VAR
	VAR
		_utfInput : REFERENCE TO WSTRING[1023];
		_sInput : REFERENCE TO STRING[255];
		_lChar1 : UDINT;
		_lChar2 : UDINT;
		_wChar1 : REFERENCE TO UINT;
		_wChar2 : REFERENCE TO UINT;
		_sOutput : REFERENCE TO STRING[255];
		_utfOutput : REFERENCE TO WSTRING[1023];
		_bChar1 : REFERENCE TO USINT;
		_iPos : INT;
		_pOutput : UDINT;
	END_VAR
END_FUNCTION_BLOCK
```

### mnTxt_History.txt
```
0.03.0	02.01.12	AH	Texte werden nun eingelesen. Das Ändern der LCID bewirkt ein Neuladen der Texte
0.04.0	10.01.12	AH	PackageVersion wird in mnTxtStatAd angezeigt
0.04.1	12.01.12	AH	Ausgabe der korrekten Anzahl vorhandener Meldungs- und Meldungs-Hilfs-Zeilen
0.04.3	17.01.12	AH	Einlesen der Meldungs- und Meldungshilfstexte hat nicht funktioniert.
0.05.0	18.01.12	AH	Texte auf 63 Zeichen verlängert. Erfordert mnParam ab Version 0.10.0
0.06.0	17.02.12	AH  Speichernutzung optimiert
0.06.1	08.02.12	AH	Bugfix
0.07.0	13.03.12	AH	Datenobjektinitialisierung wieder in den Init-Teil gelegt
0.07.1	20.03.12	AH	Abhängigkeiten ergänzt
0.08.0	22.06.12	AH	In Hilfstexten werden \n durch ein $R und $N ersetzt.
0.09.0	03.09.12	AH	Erweiterung Bug 836:Sprachresourcen können auch sprachspezifisch geladen werden.
						Konstante MNTXT_ENABLE_LANSPECRESOURCE vom Tyb USINT anlegen. 0 - Summenresourcen werden geladen, 1 - spez. Sprachresourcen
```

### Package Logical/Standard/Kanlink/KGFramework/Pkg_hlDFII - DATAFOCUS II

### Pkg_hlDFII.typ - Global data types
```iecst
(********************************************************************
 * COPYRIGHT -- Microsoft
 ********************************************************************
 * Package: pkg_sqlreq
 * File: pkg_sqlreq.typ
 * Author: hunholz
 * Created: April 05, 2011
 ********************************************************************
 * Data types of package pkg_sqlreq
 ********************************************************************)

TYPE
	hlDFIIStatAd_typ : 	STRUCT
		sPkgVersion : STRING[10];
	END_STRUCT;
	hlDFIIParMacConn_typ : 	STRUCT
		bDBservReg : USINT := 3;
		bDBservAdr : USINT := 202;
		wDBservPort : UINT := 1433;
		sServInst : STRING[15];
		sDBname : STRING[15] := 'DFII';
		wIdletimeDisconnect : UINT := 10;
	END_STRUCT;
	hlDFIIParMac_typ : 	STRUCT
		DFIIConn : hlDFIIParMacConn_typ;
		TrackConn : hlDFIIParMacConn_typ;
	END_STRUCT;
	hlDFIIPar_typ : 	STRUCT
		Mac : hlDFIIParMac_typ;
	END_STRUCT;
	IFhlDFII_typ : 	STRUCT
		In : IFhlDFII_In_typ;
		Out : IFhlDFII_Out_typ;
	END_STRUCT;
	IFhlDFII_Out_typ : 	STRUCT
		wStatus : UINT;
		xConnected : BOOL;
		xTrackConnected : BOOL;
		sStatusTracking : STRING[127];
		RespProgByCat : IFhlDFII_Out_RespProgByCat_typ;
		RespMsgEvt : IFhlDFII_Out_RespMsgEvt_typ;
		RespCntBatchEvt : IFhlDFII_Out_RespCntBatchEvt_typ;
		RespCntCntEvt : IFhlDFII_Out_RespCntCntEvt_typ;
		RespCntTimEvt : IFhlDFII_Out_RespCntTimEvt_typ;
		RespCntDosEvt : IFhlDFII_Out_RespCntDosEvt_typ;
	END_STRUCT;
	IFhlDFII_Out_RespProgByCat_typ : 	STRUCT
		wResponse : UINT; (*0 - idle, 1 - req num OK, 2 - req alpha OK, 65535 - busy*)
		bProgramNo : USINT;
		sProgramName : STRING[31];
		sCategoryName : STRING[31];
		wLoadrate : UINT;
		rSoilfactor : REAL;
		wColorIdxFor : UINT;
		wColorIdxBack : UINT;
	END_STRUCT;
	IFhlDFII_Out_RespMsgEvt_typ : 	STRUCT
		wResponse : UINT; (*0 - idle, 1 - req OK, 65535 - busy*)
	END_STRUCT;
	IFhlDFII_Out_RespCntBatchEvt_typ : 	STRUCT
		wResponse : UINT; (*0 - idle, 1 - req, OK, 65535 - busy*)
	END_STRUCT;
	IFhlDFII_Out_RespCntCntEvt_typ : 	STRUCT
		wResponse : UINT; (*0 - idle, 1 - req, OK, 65535 - busy*)
	END_STRUCT;
	IFhlDFII_Out_RespCntTimEvt_typ : 	STRUCT
		wResponse : UINT; (*0 - idle, 1 - req, OK, 65535 - busy*)
	END_STRUCT;
	IFhlDFII_Out_RespCntDosEvt_typ : 	STRUCT
		wResponse : UINT; (*0 - idle, 1 - req, OK, 65535 - busy*)
	END_STRUCT;
	IFhlDFII_In_typ : 	STRUCT
		utfMachineType : WSTRING[15];
		ReqProgByCat : IFhlDFII_In_ReqProgByCat_typ;
		ReqMsgEvt : IFhlDFII_In_ReqMsgEvt_typ;
		ReqCntBatchEvt : IFhlDFII_In_ReqCntBatchEvt_typ;
		ReqCntCntEvt : IFhlDFII_In_ReqCntCntEvt_typ;
		ReqCntTimEvt : IFhlDFII_In_ReqCntTimEvt_typ;
		ReqCntDosEvt : IFhlDFII_In_ReqCntDosEvt_typ;
		ReqUpdStatus : ARRAY[1..HLDFII_MAXIDX_REQ_UPDATESTATUS]OF IFhlDFII_In_ReqUpdStatus_typ;
		ReqUpdBatch : ARRAY[1..HLDFII_MAXIDX_REQ_UPDATEBATCH]OF IFhlDFII_In_ReqUpdBatch_typ;
	END_STRUCT;
	IFhlDFII_In_ReqProgByCat_typ : 	STRUCT
		wRequest : UINT; (*0 - idle, 1 - req num, 2 - req alpha*)
		sCategoryNo_In : STRING[11];
	END_STRUCT;
	IFhlDFII_In_ReqMsgEvt_typ : 	STRUCT
		wRequest : UINT; (*0 - idle, 1 - req*)
		bCntLines : USINT; (*1..5*)
		MsgHistList : ARRAY[1..5]OF MsgHistList_Typ;
	END_STRUCT;
	IFhlDFII_In_ReqCntBatchEvt_typ : 	STRUCT
		wRequest : UINT; (*0 - idle, 1 - request*)
		bCntLines : USINT; (*1..5*)
		CntBatchEvtList : ARRAY[1..5]OF mnCntEventBatch_Typ;
	END_STRUCT;
	IFhlDFII_In_ReqCntCntEvt_typ : 	STRUCT
		wRequest : UINT; (*0 - idle, 1 - request*)
		bCntLines : USINT; (*1..5*)
		CntCounterEvtList : ARRAY[1..5]OF mnCntEventCounter_Typ;
	END_STRUCT;
	IFhlDFII_In_ReqCntTimEvt_typ : 	STRUCT
		wRequest : UINT; (*0 - idle, 1 - request*)
		bCntLines : USINT; (*1..5*)
		CntTimerEvtList : ARRAY[1..5]OF mnCntEventTime_Typ;
	END_STRUCT;
	IFhlDFII_In_ReqCntDosEvt_typ : 	STRUCT
		wRequest : UINT; (*0 - idle, 1 - request*)
		bCntLines : USINT; (*1..5*)
		CntDosingEvtList : ARRAY[1..5]OF mnCntEventDosingId_Typ;
	END_STRUCT;
	IFhlDFII_In_ReqUpdStatus_typ : 	STRUCT
		wStatusX : UINT;
		wSubState : UINT;
		sSubState : STRING[23];
		xEnable : BOOL;
		lMachineNo : UDINT;
	END_STRUCT;
	IFhlDFII_In_ReqUpdBatch_typ : 	STRUCT
		dtTimeStamp : DATE_AND_TIME;
		lMachineNo : UDINT;
		bBatchNo : ARRAY[0..15]OF USINT;
		wLocation : UINT;
		wElement : UINT;
	END_STRUCT;
END_TYPE
```

### Pkg_hlDFII.var - Global variables
```iecst
(********************************************************************
 * COPYRIGHT -- Microsoft
 ********************************************************************
 * Package: pkg_sqlreq
 * File: pkg_sqlreq.var
 * Author: hunholz
 * Created: April 05, 2011
 ********************************************************************
 * Variables of package pkg_sqlreq
 ********************************************************************)
(*Konstanten*)
VAR CONSTANT
	HLDFII_STAT_OK : UINT := 0; (*OK*)
	HLDFII_STAT_DISABLED : UINT := 100; (*Per Konfiguration und Parameter deaktiviert*)
	HLDFII_STAT_INIT : UINT := 101; (*Initialisierung. Wartet noch auf OK von mnParam und mnEth*)
	HLDFII_STAT_NO_CONNECTION : UINT := 60000; (*Es konnte keine Verbindung zur Datenbank aufgebaut werden.*)
END_VAR
(*Stati*)
VAR
	hlDFIIStat : Stat_typ := (0);
	hlDFIIStatAd : hlDFIIStatAd_typ;
	hlDFIIPar : hlDFIIPar_typ;
	IFhlDFII : IFhlDFII_typ;
END_VAR
```

### Program Logical/Standard/Kanlink/KGFramework/Pkg_hlDFII/hlDFII (IEC) - Statemachine zur Abfrage einer SQL-Datenbank

#### hlDFIICyclic.st - Cyclic code
```iecst
(********************************************************************
 * COPYRIGHT -- Microsoft
 ********************************************************************
 * Program: hlDFII
 * File: hlDFIICyclic.st
 * Author: hunholz
 * Created: April 05, 2011
 * Changed: November 14, 2011
 ********************************************************************
 * Implementation of program hlDFII
 ********************************************************************)

PROGRAM _CYCLIC

	// Init
	IF IFmnParam.Out.xParamOK AND NOT _xInitDone THEN

		brwcsconv(ADR(_sMNo), ADR(IFmnParam.Out.utfMachineNumber), 1);

		FOR _ii := 1 TO HLDFII_MAXIDX_REQ_UPDATESTATUS DO
			_wStatusX[_ii] := 16#FFFF;
		END_FOR

		_xInitDone := TRUE;

	END_IF

	IF NOT _xReady AND IFmnEth.Out.xDataValid AND IFmnParam.Out.xParamOK AND HLDFII_RUN_CLIENT THEN

		//**********************
		// INITIALISIERUNG
		//***********************

		_CreateConnStringDFII(IP := IFmnEth.Out.IP, Conn := hlDFIIPar.Mac.DFIIConn);

		_CreateConnStringTracking(IP := IFmnEth.Out.IP, Conn := hlDFIIPar.Mac.TrackConn);

		_xReady := TRUE;

		// UDP-Log vorbereiten

		_UdpOpen.enable	 := TRUE;
		_UdpOpen.pIfAddr := 0;
		_UdpOpen.port	 := HLDFII_UDP_PORT_LOG4NET;
		_UdpOpen.options := udpOPT_BROADCAST;

	ELSIF _xReady THEN

		//***********************************
		// ZYKLISCHE ABARBEITUNG
		//***********************************

		hlDFIIStat.wStatus := 0;

		////////////////////////////////////////////////////////////////////////////////////
		////////////////////////////////////////////////////////////////////////////////////
		// DFII
		////////////////////////////////////////////////////////////////////////////////////
		////////////////////////////////////////////////////////////////////////////////////

		//*********************************************************************************
		// Request Scheduler DFII
		//*********************************************************************************

		_actReqScheduleDFII;

		//*********************************************************************************
		// Aufträge ausführen
		//*********************************************************************************

		_actProcCmdDFII;

		//*********************************************************************************
		// Verbindung nach ablauf der Idletime abbauen, wenn keine Aktion ist
		//*********************************************************************************

		IF _eStep = eSQLREQ_STEP_ERROR THEN

			_eStep := eSQLREQ_STEP_DISCONNECT;

		ELSIF (_eCmdDFIIStep = eCMD_SQLREQ_IDLE) AND(_eStep = eSQLREQ_STEP_WAITFORCOMMAND) THEN

			_GTCurrent(enable := TRUE);

			IF _GTCurrent.DT1 > _GTlastAction.DT1 THEN

				IF DiffDT(_GTCurrent.DT1, _GTlastAction.DT1) > hlDFIIPar.Mac.DFIIConn.wIdletimeDisconnect THEN

					// Idletime abgelaufen, Verbindung abbauen
					_eStep := eSQLREQ_STEP_DISCONNECT;

				END_IF

			END_IF

		ELSE

			_GTlastAction(enable := TRUE);

		END_IF

		//*********************************************************************************
		// Verbindung bei Bedarf aufbauen
		//*********************************************************************************

		IF _eCmdDFIIStep <> eCMD_SQLREQ_IDLE AND _eStep = eSQLREQ_STEP_STOP THEN

			_eStep := eSQLREQ_STEP_CONNECT;

		END_IF

		//*********************************************************************************
		// SQL-Befehle ausführen
		//*********************************************************************************

		_actProcSQLDFII;

		// Wenn Maschinenregistrierung fehlerhaft war, wiederholen nach ca. 1 Minute
		TONrepReg(IN := _bEventRegMach = 255, PT := T#60s);
		IF TONrepReg.Q THEN
			_bEventRegMach := 1;
		END_IF
		// Wenn Zeit lesen fehlerhaft war, wiederholen nach ca. 1 Minute
		TONrepGettime(IN := _bEventGetTime = 255, PT := T#60s);
		IF TONrepGettime.Q THEN
			_bEventGetTime := 1;
		END_IF

		////////////////////////////////////////////////////////////////////////////////////
		////////////////////////////////////////////////////////////////////////////////////
		// TRACKING
		////////////////////////////////////////////////////////////////////////////////////
		////////////////////////////////////////////////////////////////////////////////////

		//*********************************************************************************
		// Request Scheduler Tracking
		//*********************************************************************************

		_actReqScheduleTrack;

		//*********************************************************************************
		// Aufträge ausführen
		//*********************************************************************************

		_actProcCmdTrack;

		//*********************************************************************************
		// Verbindung nach ablauf der Idletime abbauen, wenn keine Aktion ist
		//*********************************************************************************

		IF _eTrackStep = eSQLREQ_STEP_ERROR THEN

			_eTrackStep := eSQLREQ_STEP_DISCONNECT;

		ELSIF (_eCmdTrackStep = eCMD_SQLREQ_IDLE) AND(_eTrackStep = eSQLREQ_STEP_WAITFORCOMMAND) THEN

			_GTCurrent(enable := TRUE);

			IF _GTCurrent.DT1 > _GTlastActionTrack.DT1 THEN

				IF DiffDT(_GTCurrent.DT1, _GTlastActionTrack.DT1) > hlDFIIPar.Mac.TrackConn.wIdletimeDisconnect THEN

					// Idletime abgelaufen, Verbindung abbauen
					_eTrackStep := eSQLREQ_STEP_DISCONNECT;

				END_IF

			END_IF

		ELSE

			_GTlastActionTrack(enable := TRUE);

		END_IF

		//*********************************************************************************
		// Verbindung bei Bedarf aufbauen
		//*********************************************************************************

		IF _eCmdTrackStep <> eCMD_SQLREQ_IDLE AND _eTrackStep = eSQLREQ_STEP_STOP THEN

			_eTrackStep := eSQLREQ_STEP_CONNECT;

		END_IF

		_actProcSQLTrack;

		// Wenn Zeit lesen fehlerhaft war, wiederholen nach ca. 1 Minute
		TONrepGettimeTrack(IN := _bEventGetTrackTime = _HLDFII_REQ_FAULT, PT := T#60s);
		IF TONrepGettimeTrack.Q THEN
			_bEventGetTrackTime := _HLDFII_REQ_START;
		END_IF

		//**********************************************************************************
		// UDP Logging
		//**********************************************************************************

		CASE _wStepUdp OF

			0:
				_UdpOpen();
				IF _UdpOpen.status = ERR_OK THEN
					_wStepUdp := 1;
				END_IF

			1:
				_ReadRB(wPtrWrite := _wPtrRBwrite, wPtrStart := _wPtrRBstart, wPtrRead := _wPtrRBread);

				IF _ReadRB.wStatus = ERR_OK THEN
					_wStepUdp := 2;
					_UdpSend.enable := TRUE;
					_UdpSend.ident := _UdpOpen.ident;
					_UdpSend.pHost := ADR(_CreateConnStringDFII.HostString);
					_UdpSend.port := HLDFII_UDP_PORT_LOG4NET;
					_UdpSend.pData := ADR(_sLogEntry);
					_UdpSend.datalen := SIZEOF(_sLogEntry);
				END_IF

			2:
				_UdpSend();
				IF _UdpSend.status <> ERR_FUB_BUSY THEN
					_wStepUdp := 1;
				END_IF

		END_CASE

		hlDFIIStat.wStatus := SEL(IFhlDFII.Out.xConnected,HLDFII_STAT_NO_CONNECTION, HLDFII_STAT_OK);
		IFhlDFII.Out.wStatus := SEL(IFhlDFII.Out.xConnected,HLDFII_STAT_NO_CONNECTION, HLDFII_STAT_OK);

	ELSE

		IF IFmnEth.Out.xDataValid AND IFmnParam.Out.xParamOK THEN

			hlDFIIStat.wStatus := HLDFII_STAT_DISABLED;
			IFhlDFII.Out.wStatus := HLDFII_STAT_DISABLED;

		ELSE

			hlDFIIStat.wStatus := HLDFII_STAT_INIT;
			IFhlDFII.Out.wStatus := HLDFII_STAT_INIT;

		END_IF

	END_IF

	// Debughilfe für _sSQLstring
	_wStartDebug := LIMIT(0,_wStartDebug, 992);
	_sDebugSQLstring ACCESS (ADR(_sSQLBatchEventString)+_wStartDebug);

END_PROGRAM
```

#### hlDFIIInit.st - Initialization code
```iecst
(********************************************************************
 * COPYRIGHT -- Microsoft
 ********************************************************************
 * Program: hlDFII
 * File: hlDFIIInit.st
 * Author: hunholz
 * Created: April 05, 2011
 ********************************************************************
 * Implementation of program hlDFII
 ********************************************************************)

PROGRAM _INIT

	// Packet-Version auslesen mit MO_ver aus SYS_lib und für den Additional Status zur Verfügung stellen

	_sPkgName := 'hlDFII';

	IF ( MO_ver(ADR(_sPkgName), 0, ADR(_VerStruc)) = 0 ) THEN

		brsmemcpy(ADR(hlDFIIStatAd.sPkgVersion), ADR(_VerStruc.version), SIZEOF(_VerStruc.version));

	ELSE

		hlDFIIStatAd.sPkgVersion := '---';

	END_IF

	// Init

	_xInitDone := FALSE;
	_xReady := FALSE;

	_eStep := eSQLREQ_STEP_STOP;
	_eTrackStep := eSQLREQ_STEP_STOP;

	_eCmdDFIIStep := eCMD_SQLREQ_IDLE;
	_eCmdTrackStep := eCMD_SQLREQ_IDLE;

	_bEventRegMach := _HLDFII_REQ_START;
	_bEventGetTime := _HLDFII_REQ_START;

	_bEventGetTrackTime := _HLDFII_REQ_START;

	_lConnectionIdent := 0;
	_lConnectionTrackIdent := 0;

	_wScheduleStep := _HLDFII_SCHEDSTEP_GETTIME;
	_wScheduleTrackStep := _HLDFII_SCHEDSTEP_T_GETTIME;

	_GTlastAction(enable := TRUE);
	_GTlastActionTrack(enable := TRUE);

	brsmemset(ADR(hlDFIIStat),0,SIZEOF(hlDFIIStat));

	// Create Log
	//****************************************************************************************************************
	// Log erzeugen
	//****************************************************************************************************************

	_kgArLogWrite.enable := TRUE;
	_kgArLogWrite.ident := 0;
	_kgArLogWrite.errornr := 50010;

	_kgArLogWriteTrack.enable := TRUE;
	_kgArLogWriteTrack.ident := 0;
	_kgArLogWriteTrack.errornr := 50010;

	_AsArLogCreate(enable := TRUE, pName := ADR('hlDFIIL'), len := 4096*4, memType := arlogUSRROM);

	IF _AsArLogCreate.status = ERR_OK THEN

		_kgArLogWrite.ident := _AsArLogCreate.ident;
		_kgArLogWriteTrack.ident := _AsArLogCreate.ident;

	ELSIF _AsArLogCreate.status = arlogERR_EXISTING THEN

		_AsArLogGetInfo(enable := TRUE, pName := ADR('hlDFIIL'));

		IF _AsArLogGetInfo.status = ERR_OK THEN

			_kgArLogWrite.ident := _AsArLogGetInfo.ident;
			_kgArLogWriteTrack.ident := _AsArLogCreate.ident;

		END_IF

	END_IF

	//****************************************************************************************************************
	// Ringbuffer for Logs
	//****************************************************************************************************************

	_kgRBcreateDFIIlog(sName := '_dfiilogrb', bMemType := doTEMP, wCntEntry := 10, lLenEntry := SIZEOF(_sLogEntry), wPtrWrite := _wPtrRBwrite, wPtrRead := _wPtrRBread, wPtrStart := _wPtrRBstart);

	IF _kgRBcreateDFIIlog.wStatus = ERR_OK THEN

		_wPtrRBloc := 0;

		_xRBReady := TRUE;

		_InsertRB.doIdent := _kgRBcreateDFIIlog.doIdent;
		_InsertRB.doLen := _kgRBcreateDFIIlog.doLen;
		_InsertRB.lLenEntry := SIZEOF(_sLogEntry);
		_InsertRB.pEntry := ADR(_sLogEntryI);

		_InsertRBT.doIdent := _kgRBcreateDFIIlog.doIdent;
		_InsertRBT.doLen := _kgRBcreateDFIIlog.doLen;
		_InsertRBT.lLenEntry := SIZEOF(_sLogEntry);
		_InsertRBT.pEntry := ADR(_sLogEntryT);

		_ReadRB.doIdent := _kgRBcreateDFIIlog.doIdent;
		_ReadRB.doLen := _kgRBcreateDFIIlog.doLen;
		_ReadRB.lLenEntry := SIZEOF(_sLogEntry);
		_ReadRB.pEntry := ADR(_sLogEntry);

	ELSE

		_kgArLogWrite.logLevel := arlogLEVEL_INFO;
		_kgArLogWrite.text := 'Create Ringbuffer: {##AttrVar1}';
		_kgArLogWrite.var1 := _kgRBcreateDFIIlog.wStatus;
		_kgArLogWrite.var2 := 0;
		_kgArLogWrite();

	END_IF

END_PROGRAM
```

#### hlDFIIExit.st - Exit code
```iecst
(********************************************************************
 * COPYRIGHT -- Microsoft
 ********************************************************************
 * Program: hlDFII
 * File: hlDFIIExit.st
 * Author: hunholz
 * Created: April 05, 2011
 * Changed: November 14, 2011
 ********************************************************************
 * Implementation of program hlDFII
 ********************************************************************)

PROGRAM _EXIT

	REPEAT
		_UdpClose(enable := TRUE, ident := _UdpOpen.ident);
		UNTIL
		_UdpClose.status <> ERR_FUB_BUSY
	END_REPEAT

	WHILE _eStep <> eSQLREQ_STEP_STOP DO

		CASE _eStep OF

			(* Beende Verbindungsaufbau, und baue dann die Verbindung wieder ab *)
			eSQLREQ_STEP_CONNECT_r:
				_DFII_Connect();
				IF _DFII_Connect.status <> ERR_FUB_BUSY THEN
					_eStep := eSQLREQ_STEP_DISCONNECT;
				END_IF

			(* Beende DFII_DBErrMsg *)
			eSQLREQ_STEP_GET_ERROR_r:
				_DFII_DBErrMsg();
				IF _DFII_DBErrMsg.status <> ERR_FUB_BUSY THEN
					_eStep := eSQLREQ_STEP_DISCONNECT;
				END_IF

			(* Beende Execute *)
			eSQLREQ_STEP_GPBC_r:
			eSQLREQ_STEP_WRMSG_r:
			eSQLREQ_STEP_WRCNTBATCHEVT_r:
			eSQLREQ_STEP_WRCNTCNTEVT_r:
			eSQLREQ_STEP_WRCNTTIMEVT_r:
			eSQLREQ_STEP_WRCNTDOSEVT_r:
			eSQLREQ_STEP_REGMACH_r:
			eSQLREQ_STEP_GETTIME_r:
				_DFII_DBExecute();
				IF _DFII_DBExecute.status <> ERR_FUB_BUSY THEN
					_eStep := eSQLREQ_STEP_DISCONNECT;
				END_IF

			(* Beende Fetch *)
			eSQLREQ_STEP_GPBC_FETCH_r:
			eSQLREQ_STEP_GETTIME_FETCH_r:
				_DFII_DBFetch();
				IF _DFII_DBFetch.status <> ERR_FUB_BUSY THEN
					_eStep := eSQLREQ_STEP_DISCONNECT;
				END_IF

			(* Bende GetVal *)
			eSQLREQ_STEP_GPBC_GETVAL_r:
			eSQLREQ_STEP_GETTIME_GETVAL_r:
				_DFII_GetData();
				IF _DFII_GetData.status <> ERR_FUB_BUSY THEN
					_eStep := eSQLREQ_STEP_DISCONNECT;
				END_IF

			(* Baue Verbindung ab *)
			eSQLREQ_STEP_DISCONNECT:

				_DFII_Disconnect.enable := TRUE;
				_DFII_Disconnect.connectionIdent := _lConnectionIdent;
				_eStep := eSQLREQ_STEP_DISCONNECT_r;

			(* Warte bis Verbindung abgebaut ist *)
			eSQLREQ_STEP_DISCONNECT_r:

				_DFII_Disconnect();

				IF _DFII_Disconnect.status <> ERR_FUB_BUSY THEN
					_eStep := eSQLREQ_STEP_STOP;
				END_IF

			eSQLREQ_STEP_ERROR:

				_eStep := eSQLREQ_STEP_DISCONNECT;

			ELSE

				_eStep := eSQLREQ_STEP_DISCONNECT;

		END_CASE

	END_WHILE

	WHILE _eTrackStep <> eSQLREQ_STEP_STOP DO

		CASE _eTrackStep OF

			(* Beende Verbindungsaufbau, und baue dann die Verbindung wieder ab *)
			eSQLREQ_STEP_CONNECT_r:
				_Track_Connect();
				IF _Track_Connect.status <> ERR_FUB_BUSY THEN
					_eTrackStep := eSQLREQ_STEP_DISCONNECT;
				END_IF

			(* Beende Track_DBErrMsg *)
			eSQLREQ_STEP_GET_ERROR_r:
				_Track_DBErrMsg();
				IF _Track_DBErrMsg.status <> ERR_FUB_BUSY THEN
					_eTrackStep := eSQLREQ_STEP_DISCONNECT;
				END_IF

			(* Beende Execute *)
			eSQLREQ_STEP_GETTIME_r:
			eSQLREQ_STEP_WRUPDSTATE_r:
			eSQLREQ_STEP_WRUPDLOC_r:
				_Track_DBExecute();
				IF _Track_DBExecute.status <> ERR_FUB_BUSY THEN
					_eTrackStep := eSQLREQ_STEP_DISCONNECT;
				END_IF

			(* Beende Fetch *)
			eSQLREQ_STEP_GETTIME_FETCH_r:
				_Track_DBFetch();
				IF _Track_DBFetch.status <> ERR_FUB_BUSY THEN
					_eTrackStep := eSQLREQ_STEP_DISCONNECT;
				END_IF

			(* Bende GetVal *)
			eSQLREQ_STEP_GETTIME_GETVAL_r:
				_Track_GetData();
				IF _Track_GetData.status <> ERR_FUB_BUSY THEN
					_eTrackStep := eSQLREQ_STEP_DISCONNECT;
				END_IF

			(* Baue Verbindung ab *)
			eSQLREQ_STEP_DISCONNECT:

				_Track_Disconnect.enable := TRUE;
				_Track_Disconnect.connectionIdent := _lConnectionTrackIdent;
				_eTrackStep := eSQLREQ_STEP_DISCONNECT_r;

			(* Warte bis Verbindung abgebaut ist *)
			eSQLREQ_STEP_DISCONNECT_r:

				_Track_Disconnect();

				IF _Track_Disconnect.status <> ERR_FUB_BUSY THEN
					_eTrackStep := eSQLREQ_STEP_STOP;
				END_IF

			eSQLREQ_STEP_ERROR:

				_eTrackStep := eSQLREQ_STEP_DISCONNECT;

			ELSE

				_eTrackStep := eSQLREQ_STEP_DISCONNECT;

		END_CASE

	END_WHILE

END_PROGRAM
```

#### hlDFII.typ - Local data types
```iecst
(********************************************************************
 * COPYRIGHT -- Microsoft
 ********************************************************************
 * Program: hlDFII
 * File: hlDFII.typ
 * Author: hunholz
 * Created: April 05, 2011
 * Changed: Novemer 14, 2011
 ********************************************************************
 * Local data types of program hlDFII
 ********************************************************************)

TYPE
	SQLREQ_STEPS_enum :
		(
		eSQLREQ_STEP_STOP := 0,
		eSQLREQ_STEP_CONNECT := 10,
		eSQLREQ_STEP_CONNECT_r,
		eSQLREQ_STEP_DISCONNECT := 20,
		eSQLREQ_STEP_DISCONNECT_r,
		eSQLREQ_STEP_WAITFORCOMMAND := 30,
		eSQLREQ_STEP_GET_ERROR := 200,
		eSQLREQ_STEP_GET_ERROR_r,
		eSQLREQ_STEP_LOGRB_ERROR,
		eSQLREQ_STEP_LOG_ERROR,
		eSQLREQ_STEP_LOG_ERROR1,
		eSQLREQ_STEP_ERROR, (*Fehler Schritt*)
		eSQLREQ_STEP_DUMMY,
		eSQLREQ_STEP_GPBC := 40,
		eSQLREQ_STEP_GPBC_r,
		eSQLREQ_STEP_GPBC_FETCH,
		eSQLREQ_STEP_GPBC_FETCH_r,
		eSQLREQ_STEP_GPBC_GETVAL,
		eSQLREQ_STEP_GPBC_GETVAL_r,
		eSQLREQ_STEP_WRMSG := 50,
		eSQLREQ_STEP_WRMSG_r,
		eSQLREQ_STEP_WRCNTBATCHEVT := 60,
		eSQLREQ_STEP_WRCNTBATCHEVT_r,
		eSQLREQ_STEP_WRCNTCNTEVT := 70,
		eSQLREQ_STEP_WRCNTCNTEVT_r,
		eSQLREQ_STEP_WRCNTTIMEVT := 80,
		eSQLREQ_STEP_WRCNTTIMEVT_r,
		eSQLREQ_STEP_WRCNTDOSEVT := 90,
		eSQLREQ_STEP_WRCNTDOSEVT_r,
		eSQLREQ_STEP_REGMACH := 100,
		eSQLREQ_STEP_REGMACH_r,
		eSQLREQ_STEP_GETTIME := 110,
		eSQLREQ_STEP_GETTIME_r,
		eSQLREQ_STEP_GETTIME_FETCH,
		eSQLREQ_STEP_GETTIME_FETCH_r,
		eSQLREQ_STEP_GETTIME_GETVAL,
		eSQLREQ_STEP_GETTIME_GETVAL_r,
		eSQLREQ_STEP_WRUPDLOC := 120,
		eSQLREQ_STEP_WRUPDLOC_r,
		eSQLREQ_STEP_WRUPDSTATE := 130,
		eSQLREQ_STEP_WRUPDSTATE_r
		);
	cmdSqlReq_enum :
		(
		eCMD_SQLREQ_IDLE := 0, (*Nichts zu tun*)
		eCMD_SQLREQ_CONNECT := 10, (*Verbinde mit SQL-Server*)
		eCMD_SQLREQ_CONNECT_w, (*Warte auf Verbindung*)
		eCMD_SQLREQ_DISCONNECT := 20, (*Baue Verbindung zum SQL-Server wieder ab*)
		eCMD_SQLREQ_DISCONNECT_w, (*Warte bis Verbindung abgebaut ist*)
		eCMD_SQLREQ_GET_PROG_BY_CAT := 30, (*Lese Programmnumer*)
		eCMD_SQLREQ_GET_PROG_BY_CAT_w, (*Warte auf Programmnummer*)
		eCMD_SQLREQ_GET_LOAD_LIMIT := 40, (*Lese Beladegrenze*)
		eCMD_SQLREQ_GET_LOAD_LIMIT_w,
		eCMD_SQLREQ_SET_BATCHHEIGHT := 50, (*Schreibe Postenhöhe*)
		eCMD_SQLREQ_SET_BATCHHEIGHT_w,
		eCMD_SQLREQ_WRITE_MSG := 60, (*Meldungsevent und Zähler schreiben*)
		eCMD_SQLREQ_WRITE_MSG_w,
		eCMD_SQLREQ_WRITE_CNTBATCHEVT := 70,
		eCMD_SQLREQ_WRITE_CNTBATCHEVT_w,
		eCMD_SQLREQ_WRITE_CNTCNTEVT := 80,
		eCMD_SQLREQ_WRITE_CNTCNTEVT_w,
		eCMD_SQLREQ_WRITE_CNTTIMEVT := 90,
		eCMD_SQLREQ_WRITE_CNTTIMEVT_w,
		eCMD_SQLREQ_WRITE_CNTDOSEVT := 100,
		eCMD_SQLREQ_WRITE_CNTDOSEVT_W,
		eCMD_SQLREQ_WRITE_REGMACH := 110,
		eCMD_SQLREQ_WRITE_REGMACH_w,
		eCMD_SQLREQ_WRITE_GETTIME := 120,
		eCMD_SQLREQ_WRITE_GETTIME_w,
		eCMD_SQLREQ_WRITE_UPDLOC := 130,
		eCMD_SQLREQ_WRITE_UPDLOC_w,
		eCMD_SQLREQ_WRITE_UPDSTATE := 140,
		eCMD_SQLREQ_WRITE_UPDSTATE_w
		);
	_CacheEntry_typ : 	STRUCT
		dtTimeStamp : DATE_AND_TIME;
		sCategory : STRING[11];
		sProgShortName : STRING[15];
		bProgram : USINT;
	END_STRUCT;
END_TYPE
```

#### hlDFII.var - Local variables
```iecst
(********************************************************************
 * COPYRIGHT -- Microsoft
 ********************************************************************
 * Program: hlDFII
 * File: hlDFII.var
 * Author: hunholz
 * Created: April 05, 2011
 ********************************************************************
 * Local variables of program hlDFII
 ********************************************************************)
VAR
	_eStep : SQLREQ_STEPS_enum;
	_eTrackStep : SQLREQ_STEPS_enum;
	_DFII_Connect : dbConnect;
	_lConnectionIdent : UDINT;
	_DFII_DBErrMsg : dbGetErrorMessage;
	_DFII_Disconnect : dbDisconnect;
	_sSQLstring : STRING[1023];
	_sMNo : STRING[15];
	_sCat : STRING[11];
	_DFII_DBExecute : dbExecuteSql;
	_DFII_DBFetch : dbFetchNextRow;
	_bCol : USINT;
	_DFII_GetData : dbGetData;
	_iProgNo : INT;
	_eCmdDFIIStep : cmdSqlReq_enum;
	_eCmdTrackStep : cmdSqlReq_enum;
	_GTlastAction : DTGetTime;
	_GTCurrent : DTGetTime;
	_wScheduleStep : UINT := 0;
	_xReady : BOOL;
	_bCntWrMsg : USINT;
	_sFunctionID : STRING[5];
	_sMsgNo : STRING[5];
	_sInstance : STRING[15];
	_sClass : STRING[3];
	_sEvent : STRING[5];
	_sTimeStamp : STRING[11];
	_sTime : STRING[11];
	_sValue : STRING[11];
	_bEventRegMach : USINT;
	_sShortName : STRING[15];
	TONrepReg : TON;
	_xInitDone : BOOL := FALSE;
END_VAR
VAR CONSTANT
	HLDFII_MSG_PROGBYCAT_ERR : UINT := 1000;
	HLDFII_MSG_MSGEVT_ERR : UINT := 1000;
	HLDFII_MSG_CNTBATCHEVT_ERR : UINT := 1000;
	HLDFII_MSG_CNTCNTEVT_ERR : UINT := 1000;
	HLDFII_MSG_CNTTIMEVT_ERR : UINT := 1000;
	HLDFII_MSG_CNTDOSEVT_ERR : UINT := 1000;
	_HLDFII_REQ_INACTIVE : USINT := 0;
	_HLDFII_REQ_START : USINT := 1;
	_HLDFII_REQ_RUN : USINT := 2;
	_HLDFII_REQ_FINISHED : USINT := 3;
	_HLDFII_REQ_FAULT : USINT := 255;
	_HLDFII_SCHEDSTEP_T_GETTIME : UINT := 0;
	_HLDFII_SCHEDSTEP_T_UPDLOC : UINT := 1;
	_HLDFII_SCHEDSTEP_T_UPDSTAT : UINT := 2;
	_HLDFII_SCHEDSTEP_T_MAX : UINT := 2;
	_HLDFII_SCHEDSTEP_GETTIME : UINT := 0;
	_HLDFII_SCHEDSTEP_REGMACHINE : UINT := 1;
	_HLDFII_SCHEDSTEP_PROGBYCAT : UINT := 2;
	_HLDFII_SCHEDSTEP_MSGEVENT : UINT := 3;
	_HLDFII_SCHEDSTEP_CNTBATCH : UINT := 4;
	_HLDFII_SCHEDSTEP_CNTCNT : UINT := 5;
	_HLDFII_SCHEDSTEP_CNTTIME : UINT := 6;
	_HLDFII_SCHEDSTEP_CNTDOS : UINT := 7;
	_HLDFII_SCHEDSTEP_MAX : UINT := 7;
END_VAR
VAR
	_bCntWrCntBatchEvt : USINT;
	_bCntWrCntCntEvt : USINT;
	_kgUSINT16toGUID : kgUSINT16toGUID;
	_sUDINT : STRING[11];
	_kgGUIDtoSTRING : kgGUIDtoSTRING;
	_mnParam_datetimetoa : mnParam_datetimetoa;
	_ii : UINT;
	_xWaitReqMsgEvtIsZero : BOOL;
	_xWaitReqProgByCatIsZero : BOOL;
	_xWaitReqCntBatchIsZero : BOOL;
	_xWaitReqCntCntIsZero : BOOL;
	_xWaitReqCntTimIsZero : BOOL;
	_xWaitReqCntDosIsZero : BOOL;
	_bEventGetTime : USINT;
	_wScheduleStepHelp : UINT;
	TONrepGettime : TON;
	_diTime : DINT;
	_DTSetTime : DTSetTime;
	_kgArLogWrite : kgArLogWrite;
	_AsArLogCreate : AsArLogCreate;
	_AsArLogGetInfo : AsArLogGetInfo;
END_VAR
VAR RETAIN
	_wPtrRBwrite : UINT;
	_wPtrRBread : UINT;
	_wPtrRBloc : UINT;
END_VAR
VAR
	_xRBReady : BOOL;
	_InsertRB : kgRBinsert;
	_ReadRB : kgRBread;
	_UdpOpen : UdpOpen;
	_wStepUdp : UINT;
	_sLogEntry : STRING[511];
	_UdpSend : UdpSend;
	_UdpClose : UdpClose;
	_sAction : STRING[31];
	_sPkgName : STRING[11];
	_VerStruc : MoVerStruc_typ;
	_sMark : STRING[31];
	_bCntWrCntTimeEvt : USINT;
	_bCntWrCntDoseEvt : USINT;
	_sDoseName : STRING[23];
END_VAR
VAR RETAIN
	_wPtrRBstart : UINT;
END_VAR
VAR
	_kgRBcreateDFIIlog : kgRBcreate;
	_sLogEntryI : STRING[511];
	_wStartDebug : UINT;
	_sDebugSQLstring : REFERENCE TO STRING[31];
	_sSQLBatchEventString : STRING[1023];
	_idxCustomer : UINT;
	_rLoadfactor : REAL;
	_diColIdxFor : DINT;
	_diColIdxBack : DINT;
	_sName : STRING[31];
	_Track_Connect : dbConnect;
	_CreateConnStringDFII : _CreateConnectionString;
	_CreateConnStringTracking : _CreateConnectionString;
	_wScheduleTrackStep : UINT;
	_bEventGetTrackTime : USINT;
	_GTlastActionTrack : DTGetTime;
	TONrepGettimeTrack : TON;
	_lConnectionTrackIdent : UDINT;
	_sLogEntryT : STRING[511];
	_InsertRBT : kgRBinsert;
	_sTrackAction : STRING[31];
	_Track_Disconnect : dbDisconnect;
	_sSQLstringTrack : STRING[1023];
	_Track_DBExecute : dbExecuteSql;
	_Track_DBFetch : dbFetchNextRow;
	_bTrackCol : USINT;
	_Track_GetData : dbGetData;
	_diTimeTrack : DINT;
	_Track_DBErrMsg : dbGetErrorMessage;
	_sTrackValue : STRING[11];
	_kgArLogWriteTrack : kgArLogWrite;
	_xReadyForRequestUpdateLocation : BOOL := TRUE;
	_xChange : BOOL;
	_dtTimeStampUpdBatch : ARRAY[1..HLDFII_MAXIDX_REQ_UPDATEBATCH] OF DATE_AND_TIME;
	_ReqUpdBatch : ARRAY[1..HLDFII_MAXIDX_REQ_UPDATEBATCH] OF IFhlDFII_In_ReqUpdBatch_typ;
	_xReadyForRequestUpdateState : BOOL := TRUE;
	_wStatusX : ARRAY[1..HLDFII_MAXIDX_REQ_UPDATESTATUS] OF UINT;
	_ReqUpdStatus : ARRAY[1..HLDFII_MAXIDX_REQ_UPDATESTATUS] OF IFhlDFII_In_ReqUpdStatus_typ;
	_wScheduleTrackStepHelp : UINT;
	_xUpdateLocationFinished : BOOL;
	_wIdxWriteUpdateLocation : UINT;
	_lBatchNo : UDINT;
	_GetBatchno : kgUSINT16toGUID;
	_TONRefreshTrack : TON;
	_wIdxWriteUpdateStatus : UINT;
	_xUpdateStatusFinished : BOOL;
	_sTrackMachineNo : STRING[15];
	_sSubState : STRING[23];
	_wSubState : ARRAY[1..HLDFII_MAXIDX_REQ_UPDATESTATUS] OF UINT;
	_sSubStates : ARRAY[1..HLDFII_MAXIDX_REQ_UPDATESTATUS] OF STRING[23];
END_VAR
```

#### _actReqScheduleTrack.st
```iecst
(********************************************************************
 * COPYRIGHT -- Herbert Kannegiesser GmbH
 ********************************************************************
 * Program: hlDFII
 * File: _actReqScheduleTrack.st
 * Author: hunholz
 * Created: June 20, 2012
 ********************************************************************
 * Implementation of program hlDFII
 ********************************************************************)

(* Process Requests for Track *)
ACTION _actReqScheduleTrack:

	// Der Scheduler wird nur ausgeführt, wenn kein SQL-Commando bearbeitet wird

	IF _eCmdTrackStep = eCMD_SQLREQ_IDLE THEN

		CASE _wScheduleTrackStep OF

			_HLDFII_SCHEDSTEP_T_GETTIME:

				// Uhrzeit holen
				IF _bEventGetTrackTime = _HLDFII_REQ_START THEN
					// Auftrag starten
					_eCmdTrackStep := eCMD_SQLREQ_WRITE_GETTIME;
					_bEventGetTrackTime := _HLDFII_REQ_RUN;
				END_IF

			_HLDFII_SCHEDSTEP_T_UPDLOC:

				IF _xUpdateStatusFinished THEN

					_xReadyForRequestUpdateState := TRUE;
					_xUpdateStatusFinished := FALSE;

				END_IF

				IF _xReadyForRequestUpdateLocation THEN

					_xChange := FALSE;

					FOR _ii := 1 TO HLDFII_MAXIDX_REQ_UPDATEBATCH DO

						IF IFhlDFII.In.ReqUpdBatch[_ii].dtTimeStamp <> _dtTimeStampUpdBatch[_ii] AND IFhlDFII.In.ReqUpdBatch[_ii].wLocation > 0 THEN

							_xChange := TRUE;
							_ReqUpdBatch := IFhlDFII.In.ReqUpdBatch;

						END_IF

					END_FOR

					IF _xChange THEN
						_eCmdTrackStep := eCMD_SQLREQ_WRITE_UPDLOC;
						_xReadyForRequestUpdateLocation := FALSE;
					END_IF

				END_IF

			_HLDFII_SCHEDSTEP_T_UPDSTAT:

				IF _xUpdateLocationFinished THEN

					_xReadyForRequestUpdateLocation := TRUE;
					_xUpdateLocationFinished := FALSE;

				END_IF

				IF _xReadyForRequestUpdateState THEN

						_xChange := FALSE;

					FOR _ii := 1 TO HLDFII_MAXIDX_REQ_UPDATESTATUS DO

						IF (IFhlDFII.In.ReqUpdStatus[_ii].wStatusX <> _wStatusX[_ii]) OR (IFhlDFII.In.ReqUpdStatus[_ii].wSubState <> _wSubState[_ii]
							OR brsstrcmp(ADR(IFhlDFII.In.ReqUpdStatus[_ii].sSubState),ADR(_sSubStates[_ii])) <> 0) AND IFhlDFII.In.ReqUpdStatus[_ii].xEnable THEN

							_xChange := TRUE;
							_ReqUpdStatus := IFhlDFII.In.ReqUpdStatus;

						END_IF

					END_FOR

					IF _xChange THEN
						_eCmdTrackStep := eCMD_SQLREQ_WRITE_UPDSTATE;
						_xReadyForRequestUpdateState := FALSE;
					END_IF

				END_IF

		END_CASE

	END_IF

END_ACTION
```
